C03585=1025.181,-73.447,-90.528,166.772,46.649,158.523
C03586=1025.175,-73.697,-90.517,166.769,46.652,158.524
C03587=1025.169,-73.946,-90.506,166.767,46.655,158.524
C03588=1025.164,-74.196,-90.495,166.763,46.657,158.524
C03589=1025.158,-74.446,-90.485,166.761,46.660,158.524
C03590=1025.152,-74.695,-90.475,166.758,46.663,158.524
C03591=1025.146,-74.945,-90.463,166.755,46.666,158.524
C03592=1025.140,-75.195,-90.452,166.752,46.669,158.525
C03593=1025.135,-75.445,-90.442,166.749,46.672,158.525
C03594=1025.129,-75.694,-90.431,166.746,46.675,158.525
C03595=1025.123,-75.944,-90.421,166.743,46.677,158.525
C03596=1025.117,-76.194,-90.411,166.740,46.680,158.525
C03597=1025.111,-76.443,-90.400,166.737,46.684,158.525
C03598=1025.105,-76.693,-90.389,166.734,46.686,158.525
C03599=1025.099,-76.943,-90.378,166.731,46.689,158.526
C03600=1025.093,-77.193,-90.368,166.728,46.692,158.526
C03601=1025.087,-77.442,-90.358,166.725,46.695,158.526
C03602=1025.082,-77.692,-90.347,166.722,46.698,158.526
C03603=1025.076,-77.942,-90.336,166.719,46.701,158.526
C03604=1025.070,-78.191,-90.326,166.717,46.703,158.526
C03605=1025.064,-78.441,-90.316,166.713,46.707,158.526
C03606=1025.059,-78.690,-90.305,166.710,46.709,158.526
C03607=1025.053,-78.940,-90.294,166.708,46.712,158.527
C03608=1025.047,-79.190,-90.284,166.704,46.715,158.527
C03609=1025.042,-79.440,-90.273,166.701,46.718,158.527
C03610=1025.035,-79.689,-90.263,166.699,46.721,158.527
C03611=1025.029,-79.940,-90.252,166.695,46.724,158.527
C03612=1025.023,-80.189,-90.242,166.692,46.726,158.527
C03613=1025.018,-80.439,-90.231,166.690,46.729,158.527
C03614=1025.011,-80.688,-90.221,166.686,46.732,158.528
C03615=1025.006,-80.938,-90.211,166.683,46.735,158.528
C03616=1025.000,-81.188,-90.201,166.680,46.738,158.528
C03617=1024.994,-81.438,-90.191,166.678,46.741,158.528
C03618=1024.988,-81.688,-90.181,166.674,46.744,158.528
C03619=1024.982,-81.937,-90.170,166.671,46.747,158.528
C03620=1024.976,-82.187,-90.160,166.668,46.750,158.528
C03621=1024.970,-82.436,-90.150,166.666,46.753,158.529
C03622=1024.964,-82.686,-90.140,166.662,46.756,158.529
C03623=1024.959,-82.936,-90.130,166.659,46.759,158.529
C03624=1024.952,-83.185,-90.120,166.657,46.762,158.529
C03625=1024.947,-83.436,-90.109,166.653,46.765,158.529
C03626=1024.941,-83.685,-90.099,166.650,46.768,158.529
C03627=1024.935,-83.935,-90.089,166.647,46.771,158.530
C03628=1024.929,-84.185,-90.079,166.645,46.774,158.530
C03629=1024.923,-84.434,-90.069,166.641,46.777,158.530
C03630=1024.915,-84.787,-90.055,166.637,46.781,158.530
C03631=1024.906,-85.139,-90.040,166.632,46.785,158.530
C03632=1024.899,-85.491,-90.026,166.629,46.790,158.531
C03633=1024.890,-85.842,-90.012,166.625,46.794,158.531
C03634=1024.884,-86.093,-90.002,166.621,46.797,158.531
C03635=1024.878,-86.342,-89.992,166.618,46.800,158.531
C03636=1024.873,-86.592,-89.981,166.616,46.803,158.531
C03637=1024.866,-86.842,-89.972,166.612,46.806,158.532
C03638=1024.861,-87.092,-89.962,166.609,46.809,158.532
C03639=1024.855,-87.342,-89.952,166.606,46.812,158.532
C03640=1024.849,-87.591,-89.941,166.603,46.814,158.532
C03641=1024.843,-87.840,-89.932,166.600,46.817,158.532
C03642=1024.838,-88.090,-89.922,166.597,46.820,158.532
C03643=1024.832,-88.340,-89.912,166.595,46.823,158.532
C03644=1024.826,-88.590,-89.902,166.591,46.826,158.532
C03645=1024.820,-88.839,-89.892,166.588,46.829,158.533
C03646=1024.815,-89.089,-89.882,166.585,46.833,158.533
C03647=1024.808,-89.339,-89.872,166.583,46.835,158.533
C03648=1024.804,-89.589,-89.862,166.579,46.838,158.533
C03649=1024.797,-89.838,-89.853,166.576,46.842,158.533
C03650=1024.792,-90.088,-89.842,166.574,46.844,158.533
C03651=1024.785,-90.338,-89.832,166.571,46.847,158.534
C03652=1024.780,-90.588,-89.822,166.567,46.850,158.534
C03653=1024.774,-90.838,-89.812,166.564,46.853,158.534
C03654=1024.769,-91.087,-89.803,166.561,46.856,158.534
C03655=1024.763,-91.337,-89.793,166.558,46.859,158.534
C03656=1024.757,-91.587,-89.783,166.555,46.862,158.534
C03657=1024.751,-91.837,-89.773,166.552,46.865,158.534
C03658=1024.747,-92.052,-89.764,166.549,46.868,158.534
C03659=1024.741,-92.268,-89.756,166.547,46.870,158.535
C03660=1024.737,-92.483,-89.747,166.545,46.873,158.535
C03661=1024.731,-92.699,-89.739,166.542,46.875,158.535
C03662=1024.727,-92.914,-89.731,166.539,46.878,158.535
C03663=1024.722,-93.129,-89.722,166.536,46.880,158.535
C03664=1024.717,-93.345,-89.714,166.534,46.883,158.535
C03665=1024.712,-93.560,-89.705,166.532,46.885,158.535
C03666=1024.706,-93.810,-89.696,166.528,46.888,158.535
C03667=1024.701,-94.060,-89.686,166.525,46.891,158.536
C03668=1024.695,-94.309,-89.676,166.523,46.894,158.536
C03669=1024.690,-94.559,-89.666,166.520,46.897,158.536
C03670=1024.683,-94.809,-89.656,166.516,46.900,158.536
C03671=1024.677,-95.059,-89.646,166.514,46.902,158.536
C03672=1024.673,-95.309,-89.637,166.510,46.905,158.536
C03673=1024.666,-95.558,-89.628,166.507,46.909,158.536
C03674=1024.661,-95.808,-89.618,166.504,46.912,158.536
C03675=1024.655,-96.058,-89.608,166.502,46.914,158.537
C03676=1024.650,-96.308,-89.598,166.498,46.918,158.537
C03677=1024.644,-96.557,-89.589,166.495,46.921,158.537
C03678=1024.639,-96.807,-89.579,166.493,46.923,158.537
C03679=1024.633,-97.057,-89.569,166.489,46.926,158.537
C03680=1024.627,-97.307,-89.559,166.486,46.929,158.537
C03681=1024.622,-97.556,-89.550,166.483,46.932,158.537
C03682=1024.616,-97.806,-89.540,166.481,46.935,158.538
C03683=1024.610,-98.056,-89.530,166.477,46.938,158.538
C03684=1024.605,-98.306,-89.522,166.474,46.941,158.538
C03685=1024.599,-98.555,-89.512,166.471,46.944,158.538
C03686=1024.593,-98.805,-89.503,166.469,46.947,158.538
C03687=1024.587,-99.054,-89.493,166.465,46.950,158.538
C03688=1024.582,-99.304,-89.483,166.462,46.953,158.538
C03689=1024.576,-99.555,-89.474,166.459,46.956,158.539
C03690=1024.570,-99.804,-89.465,166.455,46.959,158.539
C03691=1024.564,-100.054,-89.456,166.453,46.963,158.539
C03692=1024.558,-100.303,-89.446,166.450,46.966,158.539
C03693=1024.553,-100.553,-89.438,166.447,46.969,158.539
C03694=1024.546,-100.838,-89.426,166.444,46.972,158.539
C03695=1024.539,-101.125,-89.415,166.440,46.976,158.540
C03696=1024.533,-101.411,-89.405,166.436,46.979,158.540
C03697=1024.526,-101.696,-89.394,166.433,46.983,158.540
C03698=1024.521,-101.947,-89.385,166.430,46.986,158.540
C03699=1024.516,-102.196,-89.376,166.427,46.989,158.540
C03700=1024.509,-102.445,-89.366,166.425,46.992,158.541
C03701=1024.504,-102.695,-89.358,166.421,46.995,158.541
C03702=1024.498,-102.945,-89.348,166.418,46.998,158.541
C03703=1024.492,-103.194,-89.339,166.415,47.001,158.541
C03704=1024.487,-103.445,-89.329,166.412,47.004,158.541
C03705=1024.482,-103.694,-89.320,166.409,47.007,158.541
C03706=1024.476,-103.944,-89.311,166.406,47.010,158.541
C03707=1024.470,-104.194,-89.302,166.403,47.014,158.541
C03708=1024.464,-104.443,-89.293,166.400,47.017,158.542
C03709=1024.458,-104.694,-89.284,166.397,47.019,158.542
C03710=1024.453,-104.943,-89.275,166.394,47.023,158.542
C03711=1024.447,-105.193,-89.265,166.391,47.026,158.542
C03712=1024.442,-105.443,-89.256,166.388,47.029,158.542
C03713=1024.436,-105.693,-89.247,166.384,47.032,158.542
C03714=1024.430,-105.942,-89.238,166.382,47.035,158.543
C03715=1024.425,-106.193,-89.229,166.379,47.038,158.543
C03716=1024.419,-106.442,-89.220,166.375,47.041,158.543
C03717=1024.413,-106.692,-89.211,166.372,47.044,158.543
C03718=1024.408,-106.941,-89.202,166.370,47.047,158.543
C03719=1024.402,-107.191,-89.193,166.367,47.050,158.543
C03720=1024.396,-107.441,-89.184,166.363,47.053,158.543
C03721=1024.392,-107.691,-89.175,166.360,47.056,158.543
C03722=1024.385,-107.940,-89.166,166.357,47.059,158.544
C03723=1024.379,-108.190,-89.157,166.355,47.062,158.544
C03724=1024.374,-108.440,-89.148,166.352,47.066,158.544
C03725=1024.368,-108.689,-89.139,166.348,47.069,158.544
C03726=1024.362,-108.940,-89.130,166.345,47.072,158.544
C03727=1024.357,-109.189,-89.121,166.342,47.075,158.544
C03728=1024.351,-109.439,-89.112,166.339,47.078,158.545
C03729=1024.345,-109.689,-89.104,166.336,47.081,158.545
C03730=1024.340,-109.938,-89.095,166.333,47.084,158.545
C03731=1024.334,-110.189,-89.086,166.330,47.087,158.545
C03732=1024.329,-110.438,-89.077,166.327,47.091,158.545
C03733=1024.323,-110.688,-89.068,166.324,47.094,158.545
C03734=1024.317,-110.938,-89.059,166.321,47.097,158.546
C03735=1024.312,-111.187,-89.051,166.318,47.100,158.546
C03736=1024.306,-111.437,-89.041,166.315,47.103,158.546
C03737=1024.301,-111.687,-89.033,166.312,47.106,158.546
C03738=1024.295,-111.937,-89.024,166.308,47.110,158.546
C03739=1024.289,-112.187,-89.015,166.306,47.112,158.546
C03740=1024.283,-112.436,-89.007,166.303,47.116,158.546
C03741=1024.278,-112.686,-88.998,166.300,47.119,158.547
C03742=1024.272,-112.936,-88.989,166.297,47.122,158.547
C03743=1024.267,-113.186,-88.981,166.293,47.126,158.547
C03744=1024.261,-113.435,-88.972,166.291,47.128,158.547
C03745=1024.255,-113.685,-88.963,166.288,47.132,158.547
C03746=1024.250,-113.935,-88.954,166.285,47.135,158.547
C03747=1024.245,-114.185,-88.946,166.281,47.138,158.548
C03748=1024.239,-114.435,-88.937,166.278,47.141,158.548
C03749=1024.233,-114.684,-88.928,166.276,47.144,158.548
C03750=1024.228,-114.934,-88.919,166.273,47.147,158.548
C03751=1024.222,-115.184,-88.911,166.270,47.151,158.548
C03752=1024.216,-115.434,-88.903,166.266,47.154,158.548
C03753=1024.211,-115.683,-88.894,166.263,47.157,158.548
C03754=1024.205,-115.934,-88.885,166.260,47.160,158.549
C03755=1024.200,-116.184,-88.877,166.258,47.163,158.549
C03756=1024.194,-116.433,-88.869,166.254,47.166,158.549
C03757=1024.189,-116.683,-88.860,166.251,47.170,158.549
C03758=1024.182,-116.968,-88.850,166.248,47.173,158.549
C03759=1024.176,-117.253,-88.840,166.244,47.177,158.549
C03760=1024.169,-117.539,-88.830,166.241,47.180,158.550
C03761=1024.163,-117.825,-88.820,166.237,47.184,158.550
C03762=1024.157,-118.074,-88.812,166.235,47.187,158.550
C03763=1024.151,-118.324,-88.804,166.231,47.190,158.550
C03764=1024.146,-118.573,-88.796,166.228,47.193,158.550
C03765=1024.141,-118.823,-88.787,166.225,47.197,158.550
C03766=1024.135,-119.074,-88.778,166.222,47.200,158.551
C03767=1024.129,-119.323,-88.770,166.220,47.203,158.551
C03768=1024.124,-119.573,-88.762,166.216,47.206,158.551
C03769=1024.118,-119.822,-88.753,166.213,47.209,158.551
C03770=1024.113,-120.072,-88.745,166.210,47.213,158.551
C03771=1024.106,-120.322,-88.737,166.207,47.216,158.551
C03772=1024.102,-120.573,-88.729,166.204,47.219,158.552
C03773=1024.096,-120.822,-88.720,166.201,47.222,158.552
C03774=1024.091,-121.072,-88.712,166.198,47.225,158.552
C03775=1024.085,-121.321,-88.704,166.195,47.228,158.552
C03776=1024.080,-121.571,-88.696,166.192,47.232,158.552
C03777=1024.074,-121.822,-88.687,166.189,47.235,158.552
C03778=1024.068,-122.071,-88.679,166.185,47.239,158.552
C03779=1024.063,-122.321,-88.670,166.183,47.241,158.553
C03780=1024.057,-122.570,-88.662,166.180,47.245,158.553
///RCONF 1,0,0,0,0,0,0,0,0,0,0,0,0,0,0,0,0,0,0,0,0,0,0,0
C03781=1024.052,-122.820,-88.655,166.177,47.248,158.553
C03782=1024.046,-123.070,-88.646,166.174,47.252,158.553
C03783=1024.041,-123.320,-88.638,166.170,47.255,158.553
C03784=1024.035,-123.569,-88.630,166.167,47.258,158.553
C03785=1024.029,-123.820,-88.621,166.165,47.261,158.554
C03786=1024.024,-124.069,-88.612,166.162,47.264,158.554
C03787=1024.019,-124.320,-88.605,166.159,47.268,158.554
C03788=1024.013,-124.569,-88.597,166.155,47.271,158.554
C03789=1024.008,-124.819,-88.588,166.152,47.274,158.554
C03790=1024.002,-125.068,-88.580,166.149,47.277,158.554
C03791=1023.997,-125.319,-88.573,166.147,47.281,158.555
C03792=1023.991,-125.568,-88.565,166.144,47.284,158.555
C03793=1023.985,-125.818,-88.556,166.140,47.287,158.555
C03794=1023.981,-126.068,-88.549,166.137,47.290,158.555
C03795=1023.975,-126.317,-88.541,166.134,47.294,158.555
C03796=1023.969,-126.567,-88.532,166.131,47.297,158.555
C03797=1023.963,-126.818,-88.525,166.128,47.300,158.555
C03798=1023.958,-127.068,-88.516,166.125,47.303,158.556
C03799=1023.952,-127.317,-88.508,166.123,47.307,158.556
C03800=1023.947,-127.567,-88.500,166.119,47.310,158.556
C03801=1023.941,-127.817,-88.493,166.116,47.313,158.556
C03802=1023.936,-128.066,-88.484,166.113,47.316,158.556
C03803=1023.931,-128.315,-88.476,166.111,47.319,158.556
C03804=1023.926,-128.566,-88.467,166.108,47.320,158.556
C03805=1023.923,-128.815,-88.457,166.104,47.323,158.556
C03806=1023.919,-129.065,-88.446,166.102,47.323,158.556
C03807=1023.917,-129.314,-88.435,166.099,47.325,158.556
C03808=1023.914,-129.564,-88.424,166.097,47.325,158.556
C03809=1023.912,-129.814,-88.411,166.095,47.324,158.555
C03810=1023.912,-130.064,-88.399,166.092,47.323,158.555
C03811=1023.911,-130.313,-88.386,166.090,47.322,158.554
C03812=1023.911,-130.563,-88.371,166.087,47.321,158.554
C03813=1023.911,-130.813,-88.357,166.085,47.318,158.553
C03814=1023.912,-131.063,-88.342,166.084,47.315,158.552
C03815=1023.913,-131.313,-88.326,166.082,47.312,158.552
C03816=1023.915,-131.562,-88.310,166.080,47.308,158.551
C03817=1023.918,-131.811,-88.293,166.078,47.304,158.550
C03818=1023.920,-132.062,-88.276,166.076,47.299,158.549
C03819=1023.925,-132.312,-88.258,166.075,47.294,158.548
C03820=1023.927,-132.562,-88.239,166.073,47.288,158.546
C03821=1023.933,-132.810,-88.220,166.072,47.282,158.545
C03822=1023.637,-132.837,-88.558,166.025,47.565,158.587
C03823=1023.633,-132.587,-88.577,166.026,47.571,158.588
C03824=1023.629,-132.338,-88.595,166.027,47.577,158.589
C03825=1023.625,-132.088,-88.613,166.028,47.582,158.590
C03826=1023.622,-131.838,-88.631,166.030,47.587,158.591
C03827=1023.620,-131.589,-88.648,166.032,47.591,158.592
C03828=1023.618,-131.339,-88.664,166.034,47.595,158.593
C03829=1023.617,-131.088,-88.680,166.036,47.598,158.594
C03830=1023.616,-130.839,-88.695,166.037,47.601,158.594
C03831=1023.615,-130.589,-88.709,166.039,47.603,158.595
C03832=1023.616,-130.340,-88.723,166.042,47.605,158.596
C03833=1023.617,-130.089,-88.737,166.044,47.606,158.596
C03834=1023.618,-129.839,-88.749,166.047,47.607,158.597
C03835=1023.619,-129.590,-88.762,166.049,47.608,158.597
C03836=1023.621,-129.340,-88.773,166.051,47.607,158.597
C03837=1023.624,-129.090,-88.784,166.054,47.606,158.598
C03838=1023.627,-128.841,-88.794,166.057,47.605,158.598
C03839=1023.631,-128.591,-88.805,166.060,47.603,158.598
C03840=1023.635,-128.342,-88.814,166.062,47.601,158.598
C03841=1023.641,-128.092,-88.822,166.065,47.599,158.598
C03842=1023.646,-127.842,-88.831,166.068,47.596,158.598
C03843=1023.651,-127.593,-88.839,166.071,47.592,158.597
C03844=1023.657,-127.343,-88.846,166.074,47.589,158.597
C03845=1023.662,-127.093,-88.855,166.078,47.586,158.597
C03846=1023.668,-126.843,-88.862,166.081,47.582,158.597
C03847=1023.673,-126.593,-88.870,166.084,47.579,158.597
C03848=1023.679,-126.344,-88.878,166.086,47.576,158.597
C03849=1023.684,-126.093,-88.886,166.089,47.572,158.596
C03850=1023.690,-125.844,-88.894,166.092,47.569,158.596
C03851=1023.695,-125.594,-88.902,166.095,47.566,158.596
C03852=1023.700,-125.344,-88.910,166.098,47.562,158.596
C03853=1023.706,-125.095,-88.918,166.102,47.559,158.596
C03854=1023.711,-124.845,-88.926,166.105,47.555,158.596
C03855=1023.717,-124.595,-88.934,166.108,47.552,158.596
C03856=1023.722,-124.345,-88.942,166.111,47.548,158.595
C03857=1023.728,-124.096,-88.950,166.113,47.545,158.595
C03858=1023.734,-123.846,-88.959,166.117,47.542,158.595
C03859=1023.740,-123.596,-88.967,166.120,47.539,158.595
C03860=1023.744,-123.345,-88.975,166.123,47.535,158.595
C03861=1023.750,-123.096,-88.983,166.126,47.532,158.595
C03862=1023.756,-122.846,-88.992,166.129,47.529,158.594
C03863=1023.761,-122.596,-89.000,166.132,47.526,158.594
C03864=1023.767,-122.347,-89.008,166.135,47.522,158.594
C03865=1023.772,-122.097,-89.016,166.138,47.519,158.594
C03866=1023.777,-121.847,-89.024,166.141,47.516,158.594
C03867=1023.783,-121.598,-89.032,166.144,47.513,158.594
C03868=1023.789,-121.347,-89.041,166.147,47.509,158.593
C03869=1023.794,-121.097,-89.049,166.150,47.506,158.593
C03870=1023.800,-120.848,-89.057,166.154,47.503,158.593
C03871=1023.806,-120.598,-89.066,166.157,47.500,158.593
C03872=1023.811,-120.349,-89.074,166.159,47.496,158.593
C03873=1023.816,-120.099,-89.083,166.162,47.493,158.593
C03874=1023.823,-119.849,-89.091,166.165,47.490,158.592
C03875=1023.828,-119.599,-89.099,166.168,47.487,158.592
C03876=1023.833,-119.349,-89.107,166.172,47.483,158.592
C03877=1023.838,-119.099,-89.116,166.175,47.480,158.592
C03878=1023.844,-118.850,-89.124,166.178,47.476,158.592
C03879=1023.850,-118.600,-89.132,166.181,47.473,158.592
C03880=1023.855,-118.349,-89.141,166.183,47.470,158.592
C03881=1023.861,-118.100,-89.149,166.186,47.467,158.591
C03882=1023.867,-117.850,-89.157,166.190,47.463,158.591
C03883=1023.873,-117.565,-89.167,166.194,47.459,158.591
C03884=1023.879,-117.280,-89.177,166.197,47.456,158.591
C03885=1023.885,-116.995,-89.187,166.200,47.452,158.591
C03886=1023.892,-116.709,-89.197,166.204,47.448,158.590
C03887=1023.897,-116.459,-89.205,166.207,47.445,158.590
C03888=1023.903,-116.210,-89.214,166.210,47.442,158.590
C03889=1023.909,-115.960,-89.222,166.212,47.439,158.590
C03890=1023.915,-115.710,-89.231,166.216,47.436,158.590
C03891=1023.920,-115.460,-89.239,166.219,47.432,158.590
C03892=1023.925,-115.210,-89.247,166.222,47.429,158.589
C03893=1023.931,-114.960,-89.256,166.225,47.426,158.589
C03894=1023.937,-114.711,-89.264,166.228,47.423,158.589
C03895=1023.942,-114.461,-89.273,166.231,47.419,158.589
C03896=1023.948,-114.211,-89.282,166.233,47.416,158.589
C03897=1023.954,-113.961,-89.291,166.237,47.413,158.589
C03898=1023.959,-113.712,-89.299,166.240,47.410,158.589
C03899=1023.965,-113.461,-89.308,166.243,47.406,158.588
C03900=1023.970,-113.211,-89.317,166.246,47.403,158.588
C03901=1023.975,-112.962,-89.325,166.249,47.400,158.588
C03902=1023.981,-112.712,-89.335,166.252,47.397,158.588
C03903=1023.987,-112.462,-89.343,166.255,47.393,158.588
C03904=1023.992,-112.213,-89.352,166.258,47.390,158.588
C03905=1023.999,-111.962,-89.360,166.261,47.387,158.587
C03906=1024.004,-111.713,-89.369,166.265,47.384,158.587
C03907=1024.009,-111.464,-89.378,166.268,47.381,158.587
C03908=1024.015,-111.213,-89.386,166.271,47.377,158.587
C03909=1024.021,-110.964,-89.396,166.273,47.374,158.587
C03910=1024.026,-110.714,-89.404,166.276,47.371,158.587
C03911=1024.032,-110.464,-89.413,166.280,47.368,158.587
C03912=1024.037,-110.214,-89.421,166.283,47.365,158.586
C03913=1024.043,-109.965,-89.431,166.286,47.361,158.586
C03914=1024.049,-109.715,-89.439,166.289,47.358,158.586
C03915=1024.054,-109.465,-89.448,166.291,47.355,158.586
C03916=1024.060,-109.215,-89.458,166.294,47.352,158.586
C03917=1024.065,-108.966,-89.466,166.298,47.349,158.586
C03918=1024.071,-108.716,-89.475,166.301,47.346,158.585
C03919=1024.077,-108.466,-89.484,166.304,47.342,158.585
C03920=1024.082,-108.216,-89.493,166.307,47.339,158.585
C03921=1024.088,-107.966,-89.502,166.310,47.336,158.585
C03922=1024.094,-107.717,-89.511,166.313,47.333,158.585
C03923=1024.099,-107.466,-89.519,166.316,47.330,158.585
C03924=1024.105,-107.217,-89.529,166.319,47.326,158.585
C03925=1024.111,-106.967,-89.538,166.322,47.323,158.584
C03926=1024.116,-106.718,-89.547,166.325,47.319,158.584
C03927=1024.122,-106.468,-89.555,166.329,47.316,158.584
C03928=1024.128,-106.218,-89.565,166.331,47.313,158.584
C03929=1024.133,-105.969,-89.573,166.334,47.310,158.584
C03930=1024.139,-105.719,-89.583,166.337,47.307,158.584
C03931=1024.145,-105.469,-89.591,166.341,47.304,158.583
C03932=1024.151,-105.219,-89.601,166.344,47.301,158.583
C03933=1024.155,-104.969,-89.610,166.347,47.298,158.583
C03934=1024.161,-104.719,-89.620,166.349,47.295,158.583
C03935=1024.167,-104.470,-89.628,166.352,47.291,158.583
C03936=1024.173,-104.220,-89.638,166.355,47.288,158.583
C03937=1024.178,-103.970,-89.646,166.359,47.285,158.582
C03938=1024.184,-103.720,-89.656,166.362,47.282,158.582
C03939=1024.190,-103.471,-89.665,166.364,47.279,158.582
C03940=1024.195,-103.221,-89.674,166.367,47.276,158.582
C03941=1024.201,-102.971,-89.683,166.371,47.273,158.582
C03942=1024.206,-102.721,-89.692,166.374,47.270,158.582
C03943=1024.213,-102.471,-89.702,166.377,47.266,158.582
C03944=1024.218,-102.222,-89.711,166.380,47.263,158.582
C03945=1024.224,-101.972,-89.720,166.383,47.260,158.581
C03946=1024.229,-101.722,-89.730,166.386,47.257,158.581
C03947=1024.236,-101.437,-89.740,166.390,47.253,158.581
C03948=1024.242,-101.151,-89.751,166.393,47.249,158.581
C03949=1024.249,-100.865,-89.762,166.396,47.246,158.581
C03950=1024.256,-100.579,-89.772,166.400,47.242,158.580
C03951=1024.260,-100.330,-89.781,166.402,47.239,158.580
C03952=1024.267,-100.080,-89.791,166.406,47.236,158.580
C03953=1024.273,-99.830,-89.800,166.409,47.233,158.580
C03954=1024.278,-99.581,-89.809,166.412,47.230,158.580
C03955=1024.284,-99.331,-89.819,166.415,47.227,158.580
C03956=1024.290,-99.082,-89.828,166.419,47.224,158.580
C03957=1024.295,-98.831,-89.837,166.421,47.220,158.579
C03958=1024.301,-98.581,-89.847,166.424,47.217,158.579
C03959=1024.307,-98.332,-89.856,166.427,47.214,158.579
C03960=1024.313,-98.082,-89.866,166.430,47.211,158.579
C03961=1024.319,-97.832,-89.874,166.434,47.208,158.579
C03962=1024.324,-97.582,-89.884,166.436,47.205,158.579
C03963=1024.330,-97.333,-89.894,166.439,47.202,158.578
C03964=1024.335,-97.082,-89.904,166.442,47.199,158.578
C03965=1024.341,-96.833,-89.913,166.446,47.196,158.578
C03966=1024.346,-96.583,-89.923,166.448,47.193,158.578
C03967=1024.352,-96.333,-89.933,166.451,47.190,158.578
C03968=1024.358,-96.084,-89.942,166.454,47.187,158.578
C03969=1024.363,-95.834,-89.952,166.457,47.183,158.578
C03970=1024.370,-95.584,-89.962,166.460,47.181,158.577
C03971=1024.374,-95.335,-89.972,166.463,47.177,158.577
C03972=1024.381,-95.085,-89.981,166.466,47.174,158.577
C03973=1024.386,-94.835,-89.991,166.470,47.172,158.577
C03974=1024.391,-94.585,-90.000,166.472,47.169,158.577
C03975=1024.397,-94.335,-90.010,166.475,47.166,158.577
C03976=1024.403,-94.086,-90.020,166.478,47.163,158.577
C03977=1024.408,-93.836,-90.029,166.482,47.160,158.577
C03978=1024.414,-93.587,-90.040,166.485,47.157,158.576
C03979=1024.420,-93.337,-90.050,166.487,47.154,158.576
C03980=1024.426,-93.087,-90.059,166.490,47.151,158.576
C03981=1024.431,-92.838,-90.069,166.494,47.148,158.576
C03982=1024.437,-92.588,-90.079,166.497,47.144,158.576
C03983=1024.443,-92.338,-90.088,166.499,47.142,158.576
C03984=1024.448,-92.088,-90.098,166.502,47.138,158.576
C03985=1024.454,-91.839,-90.108,166.506,47.135,158.575
C03986=1024.459,-91.589,-90.118,166.509,47.132,158.575
C03987=1024.466,-91.339,-90.127,166.511,47.129,158.575
C03988=1024.471,-91.089,-90.138,166.514,47.126,158.575
C03989=1024.477,-90.839,-90.147,166.518,47.123,158.575
C03990=1024.482,-90.590,-90.157,166.521,47.120,158.575
C03991=1024.488,-90.340,-90.166,166.523,47.117,158.574
C03992=1024.494,-90.090,-90.177,166.526,47.114,158.574
C03993=1024.500,-89.841,-90.187,166.530,47.111,158.574
C03994=1024.505,-89.590,-90.197,166.533,47.108,158.574
C03995=1024.511,-89.341,-90.206,166.535,47.105,158.574
C03996=1024.516,-89.091,-90.216,166.538,47.102,158.574
C03997=1024.523,-88.841,-90.226,166.542,47.099,158.574
C03998=1024.528,-88.592,-90.237,166.545,47.096,158.573
C03999=1024.535,-88.342,-90.246,166.548,47.093,158.573
C04000=1024.540,-88.092,-90.257,166.550,47.090,158.573
C04001=1024.546,-87.843,-90.266,166.554,47.087,158.573
C04002=1024.551,-87.593,-90.276,166.557,47.084,158.573
C04003=1024.557,-87.344,-90.286,166.560,47.081,158.573
C04004=1024.563,-87.094,-90.296,166.562,47.078,158.572
C04005=1024.569,-86.844,-90.306,166.566,47.075,158.572
C04006=1024.575,-86.594,-90.316,166.569,47.072,158.572
C04007=1024.581,-86.344,-90.326,166.572,47.068,158.572
C04008=1024.586,-86.094,-90.337,166.574,47.066,158.572
C04009=1024.593,-85.845,-90.346,166.578,47.062,158.572
C04010=1024.597,-85.595,-90.356,166.581,47.059,158.572
C04011=1024.605,-85.312,-90.368,166.584,47.056,158.571
C04012=1024.611,-85.028,-90.379,166.588,47.052,158.571
C04013=1024.618,-84.744,-90.391,166.591,47.048,158.571
C04014=1024.625,-84.460,-90.402,166.594,47.045,158.571
C04015=1024.630,-84.212,-90.412,166.598,47.042,158.571
C04016=1024.636,-83.962,-90.422,166.601,47.039,158.571
C04017=1024.642,-83.712,-90.432,166.603,47.036,158.570
C04018=1024.648,-83.462,-90.443,166.606,47.033,158.570
C04019=1024.654,-83.212,-90.452,166.610,47.030,158.570
C04020=1024.659,-82.963,-90.463,166.613,47.027,158.570
C04021=1024.666,-82.713,-90.473,166.616,47.024,158.570
C04022=1024.671,-82.463,-90.483,166.618,47.021,158.570
C04023=1024.678,-82.214,-90.493,166.621,47.017,158.569
C04024=1024.683,-81.964,-90.503,166.625,47.014,158.569
C04025=1024.689,-81.714,-90.514,166.628,47.011,158.569
C04026=1024.695,-81.464,-90.524,166.630,47.008,158.569
C04027=1024.701,-81.215,-90.533,166.633,47.005,158.569
C04028=1024.707,-80.965,-90.544,166.637,47.002,158.569
C04029=1024.713,-80.715,-90.554,166.640,46.999,158.568
C04030=1024.719,-80.466,-90.565,166.643,46.996,158.568
C04031=1024.725,-80.216,-90.574,166.645,46.993,158.568
C04032=1024.731,-79.966,-90.585,166.649,46.990,158.568
C04033=1024.737,-79.716,-90.596,166.652,46.987,158.568
C04034=1024.742,-79.466,-90.606,166.655,46.984,158.568
C04035=1024.748,-79.216,-90.617,166.657,46.981,158.567
C04036=1024.754,-78.967,-90.627,166.661,46.978,158.567
C04037=1024.760,-78.717,-90.637,166.664,46.975,158.567
C04038=1024.765,-78.467,-90.648,166.666,46.972,158.567
C04039=1024.773,-78.159,-90.661,166.670,46.969,158.567
C04040=1024.779,-77.850,-90.674,166.673,46.965,158.567
C04041=1024.786,-77.541,-90.687,166.678,46.962,158.567
C04042=1024.794,-77.232,-90.700,166.682,46.957,158.566
C04043=1024.800,-76.983,-90.710,166.684,46.955,158.566
C04044=1024.806,-76.734,-90.721,166.687,46.952,158.566
C04045=1024.811,-76.484,-90.731,166.690,46.948,158.566
C04046=1024.817,-76.234,-90.742,166.693,46.946,158.566
C04047=1024.823,-75.984,-90.753,166.696,46.943,158.566
C04048=1024.830,-75.734,-90.763,166.700,46.940,158.566
C04049=1024.835,-75.485,-90.774,166.703,46.937,158.565
C04050=1024.841,-75.235,-90.785,166.705,46.934,158.565
C04051=1024.847,-74.985,-90.795,166.708,46.931,158.565
C04052=1024.852,-74.735,-90.806,166.712,46.928,158.565
C04053=1024.858,-74.486,-90.817,166.714,46.925,158.565
C04054=1024.865,-74.236,-90.827,166.717,46.922,158.565
C04055=1024.871,-73.987,-90.838,166.720,46.919,158.564
C04056=1024.876,-73.736,-90.849,166.723,46.916,158.564
C04057=1024.881,-73.487,-90.860,166.726,46.914,158.564
C04058=1024.887,-73.237,-90.871,166.729,46.911,158.564
C04059=1024.893,-72.988,-90.882,166.732,46.908,158.564
C04060=1024.899,-72.738,-90.892,166.735,46.906,158.564
C04061=1024.904,-72.489,-90.903,166.737,46.903,158.564
C04062=1024.911,-72.239,-90.915,166.741,46.900,158.564
C04063=1024.916,-71.989,-90.925,166.744,46.897,158.563
C04064=1024.922,-71.740,-90.936,166.746,46.894,158.563
C04065=1024.928,-71.490,-90.947,166.750,46.891,158.563
C04066=1024.932,-71.240,-90.958,166.753,46.888,158.563
C04067=1024.939,-70.989,-90.969,166.755,46.886,158.563
C04068=1024.945,-70.740,-90.980,166.758,46.882,158.563
C04069=1024.950,-70.490,-90.991,166.761,46.880,158.563
C04070=1024.956,-70.241,-91.002,166.764,46.877,158.562
C04071=1024.961,-70.005,-91.012,166.767,46.874,158.562
C04072=1024.967,-69.769,-91.022,166.770,46.872,158.562
C04073=1024.972,-69.533,-91.033,166.772,46.869,158.562
C04074=1024.978,-69.296,-91.044,166.775,46.866,158.562
C04075=1024.983,-69.060,-91.054,166.778,46.864,158.562
C04076=1024.989,-68.824,-91.064,166.781,46.861,158.562
C04077=1024.994,-68.588,-91.075,166.784,46.859,158.562
C04078=1024.999,-68.352,-91.085,166.787,46.856,158.562
C04079=1025.006,-68.103,-91.097,166.789,46.853,158.561
C04080=1025.012,-67.853,-91.108,166.793,46.850,158.561
C04081=1025.018,-67.604,-91.119,166.795,46.847,158.561
C04082=1025.023,-67.354,-91.130,166.798,46.845,158.561
C04083=1025.030,-67.104,-91.141,166.802,46.842,158.561
C04084=1025.035,-66.855,-91.152,166.804,46.839,158.561
C04085=1025.040,-66.605,-91.164,166.807,46.836,158.560
C04086=1025.046,-66.355,-91.175,166.810,46.833,158.560
C04087=1025.052,-66.105,-91.186,166.813,46.830,158.560
C04088=1025.058,-65.856,-91.197,166.816,46.827,158.560
C04089=1025.064,-65.606,-91.208,166.818,46.825,158.560
C04090=1025.071,-65.356,-91.219,166.822,46.821,158.560
///RCONF 1,0,0,1,0,0,0,0,0,0,0,0,0,0,0,0,0,0,0,0,0,0,0,0
C04091=1025.076,-65.107,-91.230,166.825,46.818,158.560
C04092=1025.081,-64.857,-91.242,166.827,46.816,158.560
C04093=1025.088,-64.607,-91.253,166.831,46.813,158.559
C04094=1025.093,-64.358,-91.264,166.834,46.810,158.559
C04095=1025.099,-64.108,-91.275,166.836,46.807,158.559
C04096=1025.106,-63.858,-91.286,166.839,46.804,158.559
C04097=1025.112,-63.609,-91.298,166.843,46.801,158.559
C04098=1025.117,-63.359,-91.309,166.845,46.799,158.559
C04099=1025.123,-63.109,-91.320,166.848,46.796,158.558
C04100=1025.129,-62.859,-91.331,166.851,46.793,158.558
C04101=1025.135,-62.610,-91.343,166.854,46.790,158.558
C04102=1025.141,-62.360,-91.354,166.857,46.787,158.558
C04103=1025.147,-62.111,-91.365,166.859,46.784,158.558
C04104=1025.153,-61.861,-91.376,166.863,46.781,158.558
C04105=1025.158,-61.612,-91.388,166.866,46.779,158.558
C04106=1025.165,-61.361,-91.400,166.869,46.776,158.557
C04107=1025.170,-61.112,-91.411,166.872,46.773,158.557
C04108=1025.176,-60.862,-91.421,166.875,46.770,158.557
C04109=1025.183,-60.613,-91.433,166.877,46.767,158.557
C04110=1025.189,-60.363,-91.444,166.881,46.764,158.557
C04111=1025.194,-60.113,-91.456,166.883,46.761,158.557
C04112=1025.200,-59.864,-91.468,166.886,46.758,158.556
C04113=1025.207,-59.614,-91.479,166.890,46.756,158.556
C04114=1025.212,-59.364,-91.490,166.892,46.753,158.556
C04115=1025.219,-59.115,-91.502,166.895,46.750,158.556
C04116=1025.224,-58.865,-91.513,166.898,46.747,158.556
C04117=1025.230,-58.615,-91.524,166.901,46.744,158.556
C04118=1025.236,-58.366,-91.536,166.904,46.741,158.555
C04119=1025.243,-58.116,-91.547,166.907,46.738,158.555
C04120=1025.248,-57.866,-91.558,166.909,46.735,158.555
C04121=1025.255,-57.617,-91.570,166.913,46.732,158.555
C04122=1025.260,-57.367,-91.582,166.915,46.729,158.555
C04123=1025.266,-57.117,-91.593,166.918,46.727,158.555
C04124=1025.272,-56.868,-91.604,166.922,46.724,158.555
C04125=1025.279,-56.618,-91.616,166.924,46.721,158.554
C04126=1025.285,-56.369,-91.627,166.927,46.718,158.554
C04127=1025.290,-56.118,-91.639,166.930,46.715,158.554
C04128=1025.297,-55.869,-91.651,166.933,46.712,158.554
C04129=1025.303,-55.619,-91.662,166.936,46.709,158.554
C04130=1025.309,-55.370,-91.674,166.939,46.706,158.554
C04131=1025.315,-55.120,-91.685,166.941,46.703,158.553
C04132=1025.320,-54.870,-91.696,166.945,46.700,158.553
C04133=1025.327,-54.621,-91.708,166.947,46.697,158.553
C04134=1025.333,-54.370,-91.719,166.950,46.694,158.553
C04135=1025.339,-54.122,-91.731,166.954,46.691,158.553
C04136=1025.346,-53.871,-91.742,166.956,46.688,158.552
C04137=1025.351,-53.622,-91.754,166.959,46.686,158.552
C04138=1025.357,-53.372,-91.766,166.963,46.683,158.552
C04139=1025.364,-53.092,-91.779,166.966,46.679,158.552
C04140=1025.372,-52.812,-91.792,166.969,46.676,158.552
C04141=1025.378,-52.532,-91.805,166.972,46.673,158.552
C04142=1025.384,-52.252,-91.818,166.975,46.669,158.551
C04143=1025.391,-52.001,-91.830,166.978,46.666,158.551
C04144=1025.397,-51.752,-91.842,166.981,46.663,158.551
C04145=1025.403,-51.503,-91.853,166.984,46.660,158.551
C04146=1025.410,-51.253,-91.864,166.987,46.657,158.551
C04147=1025.416,-51.003,-91.877,166.989,46.655,158.550
C04148=1025.421,-50.753,-91.888,166.993,46.651,158.550
C04149=1025.427,-50.504,-91.900,166.995,46.649,158.550
C04150=1025.434,-50.254,-91.912,166.998,46.646,158.550
C04151=1025.439,-50.004,-91.924,167.001,46.643,158.550
C04152=1025.446,-49.755,-91.936,167.004,46.641,158.550
C04153=1025.452,-49.505,-91.948,167.006,46.638,158.550
C04154=1025.457,-49.256,-91.961,167.010,46.635,158.549
C04155=1025.464,-49.006,-91.972,167.013,46.632,158.549
C04156=1025.469,-48.756,-91.984,167.016,46.630,158.549
C04157=1025.475,-48.507,-91.996,167.019,46.627,158.549
C04158=1025.481,-48.257,-92.008,167.021,46.624,158.549
C04159=1025.486,-48.008,-92.021,167.025,46.622,158.549
C04160=1025.493,-47.758,-92.033,167.027,46.619,158.549
C04161=1025.499,-47.507,-92.044,167.030,46.616,158.548
C04162=1025.505,-47.258,-92.056,167.032,46.613,158.548
C04163=1025.511,-47.009,-92.069,167.036,46.611,158.548
C04164=1025.516,-46.759,-92.081,167.038,46.608,158.548
C04165=1025.523,-46.509,-92.093,167.041,46.605,158.548
C04166=1025.528,-46.260,-92.105,167.044,46.602,158.548
C04167=1025.535,-46.011,-92.117,167.047,46.600,158.548
C04168=1025.541,-45.761,-92.130,167.049,46.597,158.547
C04169=1025.546,-45.511,-92.141,167.053,46.594,158.547
C04170=1025.553,-45.261,-92.153,167.055,46.591,158.547
C04171=1025.559,-45.011,-92.166,167.058,46.588,158.547
C04172=1025.565,-44.762,-92.178,167.061,46.586,158.547
C04173=1025.571,-44.513,-92.190,167.064,46.583,158.547
C04174=1025.576,-44.263,-92.202,167.067,46.580,158.546
C04175=1025.583,-44.013,-92.214,167.070,46.577,158.546
C04176=1025.589,-43.763,-92.227,167.073,46.575,158.546
C04177=1025.594,-43.514,-92.239,167.075,46.572,158.546
C04178=1025.601,-43.265,-92.251,167.079,46.569,158.546
C04179=1025.607,-43.015,-92.264,167.081,46.566,158.546
C04180=1025.613,-42.765,-92.276,167.084,46.563,158.545
C04181=1025.619,-42.515,-92.288,167.087,46.561,158.545
C04182=1025.625,-42.266,-92.300,167.090,46.558,158.545
C04183=1025.631,-42.016,-92.312,167.092,46.555,158.545
C04184=1025.637,-41.767,-92.325,167.095,46.552,158.545
C04185=1025.643,-41.517,-92.337,167.098,46.549,158.545
C04186=1025.650,-41.267,-92.349,167.101,46.547,158.545
C04187=1025.655,-41.018,-92.362,167.103,46.544,158.544
C04188=1025.661,-40.768,-92.374,167.107,46.541,158.544
C04189=1025.668,-40.518,-92.386,167.109,46.538,158.544
C04190=1025.674,-40.269,-92.399,167.112,46.535,158.544
C04191=1025.679,-40.019,-92.411,167.116,46.532,158.544
C04192=1025.686,-39.769,-92.423,167.118,46.530,158.544
C04193=1025.692,-39.519,-92.436,167.121,46.527,158.543
C04194=1025.698,-39.271,-92.448,167.124,46.524,158.543
C04195=1025.704,-39.021,-92.461,167.127,46.521,158.543
C04196=1025.710,-38.771,-92.473,167.129,46.519,158.543
C04197=1025.716,-38.521,-92.486,167.133,46.516,158.543
C04198=1025.722,-38.271,-92.498,167.135,46.513,158.543
C04199=1025.728,-38.022,-92.511,167.137,46.511,158.542
C04200=1025.734,-37.772,-92.524,167.141,46.508,158.542
C04201=1025.739,-37.523,-92.536,167.143,46.506,158.542
C04202=1025.745,-37.273,-92.549,167.146,46.503,158.542
C04203=1025.753,-36.993,-92.563,167.150,46.500,158.542
C04204=1025.759,-36.713,-92.577,167.153,46.496,158.542
C04205=1025.766,-36.433,-92.592,167.155,46.494,158.541
C04206=1025.773,-36.154,-92.606,167.158,46.491,158.541
C04207=1025.779,-35.904,-92.618,167.162,46.488,158.541
C04208=1025.785,-35.654,-92.631,167.164,46.486,158.541
C04209=1025.791,-35.404,-92.644,167.167,46.482,158.541
C04210=1025.798,-35.155,-92.656,167.170,46.480,158.541
C04211=1025.803,-34.906,-92.669,167.173,46.477,158.541
C04212=1025.809,-34.656,-92.681,167.175,46.475,158.540
C04213=1025.815,-34.407,-92.694,167.179,46.472,158.540
C04214=1025.821,-34.157,-92.707,167.181,46.469,158.540
C04215=1025.827,-33.907,-92.719,167.183,46.467,158.540
C04216=1025.833,-33.658,-92.733,167.187,46.464,158.540
C04217=1025.839,-33.408,-92.745,167.189,46.461,158.540
C04218=1025.845,-33.159,-92.758,167.193,46.459,158.539
C04219=1025.851,-32.909,-92.771,167.195,46.456,158.539
C04220=1025.857,-32.659,-92.784,167.198,46.453,158.539
C04221=1025.863,-32.410,-92.797,167.200,46.450,158.539
C04222=1025.869,-32.160,-92.809,167.204,46.448,158.539
C04223=1025.876,-31.911,-92.822,167.206,46.445,158.539
C04224=1025.882,-31.661,-92.835,167.209,46.442,158.538
C04225=1025.888,-31.411,-92.847,167.212,46.439,158.538
C04226=1025.894,-31.162,-92.860,167.214,46.437,158.538
C04227=1025.900,-30.912,-92.873,167.217,46.434,158.538
C04228=1025.906,-30.663,-92.886,167.220,46.431,158.538
C04229=1025.912,-30.413,-92.899,167.223,46.428,158.538
C04230=1025.918,-30.164,-92.912,167.226,46.426,158.538
C04231=1025.924,-29.914,-92.925,167.229,46.423,158.537
C04232=1025.930,-29.665,-92.938,167.231,46.420,158.537
C04233=1025.936,-29.415,-92.950,167.234,46.417,158.537
C04234=1025.943,-29.165,-92.964,167.237,46.414,158.537
C04235=1025.948,-28.916,-92.976,167.240,46.412,158.537
C04236=1025.955,-28.666,-92.990,167.242,46.409,158.536
C04237=1025.961,-28.416,-93.002,167.245,46.406,158.536
C04238=1025.967,-28.166,-93.016,167.248,46.403,158.536
C04239=1025.973,-27.917,-93.028,167.250,46.401,158.536
C04240=1025.980,-27.668,-93.041,167.254,46.398,158.536
C04241=1025.986,-27.418,-93.054,167.256,46.396,158.536
C04242=1025.992,-27.168,-93.067,167.259,46.393,158.535
C04243=1025.998,-26.919,-93.081,167.262,46.390,158.535
C04244=1026.004,-26.669,-93.093,167.264,46.388,158.535
C04245=1026.010,-26.420,-93.106,167.267,46.385,158.535
C04246=1026.016,-26.170,-93.120,167.270,46.383,158.535
C04247=1026.021,-25.920,-93.133,167.273,46.380,158.535
C04248=1026.028,-25.671,-93.146,167.275,46.377,158.534
C04249=1026.034,-25.422,-93.159,167.278,46.375,158.534
C04250=1026.040,-25.172,-93.172,167.281,46.372,158.534
C04251=1026.046,-24.922,-93.186,167.283,46.369,158.534
C04252=1026.052,-24.672,-93.200,167.287,46.367,158.534
C04253=1026.058,-24.423,-93.213,167.289,46.364,158.534
C04254=1026.064,-24.173,-93.225,167.291,46.361,158.533
C04255=1026.070,-23.924,-93.239,167.295,46.359,158.533
C04256=1026.076,-23.674,-93.252,167.297,46.356,158.533
C04257=1026.082,-23.425,-93.266,167.300,46.353,158.533
C04258=1026.088,-23.175,-93.278,167.303,46.351,158.533
C04259=1026.095,-22.925,-93.292,167.305,46.348,158.533
C04260=1026.101,-22.676,-93.305,167.309,46.345,158.533
C04261=1026.106,-22.426,-93.319,167.311,46.343,158.532
C04262=1026.112,-22.176,-93.332,167.313,46.340,158.532
C04263=1026.119,-21.927,-93.345,167.317,46.337,158.532
C04264=1026.125,-21.678,-93.358,167.319,46.335,158.532
C04265=1026.131,-21.428,-93.372,167.322,46.332,158.532
C04266=1026.137,-21.178,-93.386,167.325,46.329,158.532
C04267=1026.144,-20.898,-93.400,167.328,46.326,158.531
C04268=1026.151,-20.617,-93.415,167.331,46.323,158.531
C04269=1026.158,-20.337,-93.430,167.334,46.320,158.531
C04270=1026.165,-20.055,-93.446,167.337,46.317,158.531
C04271=1026.171,-19.806,-93.459,167.340,46.314,158.531
C04272=1026.177,-19.556,-93.472,167.342,46.312,158.530
C04273=1026.182,-19.307,-93.486,167.345,46.310,158.530
C04274=1026.189,-19.057,-93.499,167.348,46.307,158.530
C04275=1026.195,-18.807,-93.513,167.350,46.304,158.530
C04276=1026.202,-18.558,-93.526,167.353,46.301,158.530
C04277=1026.207,-18.309,-93.540,167.356,46.299,158.530
C04278=1026.213,-18.059,-93.553,167.358,46.296,158.529
C04279=1026.220,-17.809,-93.567,167.362,46.293,158.529
C04280=1026.226,-17.560,-93.580,167.364,46.290,158.529
C04281=1026.232,-17.311,-93.594,167.367,46.288,158.529
C04282=1026.238,-17.061,-93.607,167.370,46.285,158.529
C04283=1026.245,-16.811,-93.621,167.372,46.282,158.529
C04284=1026.251,-16.562,-93.634,167.375,46.279,158.528
C04285=1026.256,-16.312,-93.647,167.378,46.277,158.528
C04286=1026.263,-16.062,-93.661,167.380,46.274,158.528
C04287=1026.269,-15.813,-93.674,167.383,46.271,158.528
C04288=1026.275,-15.563,-93.688,167.386,46.269,158.528
C04289=1026.281,-15.314,-93.702,167.388,46.267,158.528
C04290=1026.287,-15.064,-93.716,167.391,46.264,158.527
C04291=1026.293,-14.815,-93.729,167.394,46.261,158.527
C04292=1026.299,-14.565,-93.743,167.396,46.259,158.527
C04293=1026.306,-14.315,-93.757,167.400,46.256,158.527
C04294=1026.311,-14.066,-93.771,167.402,46.254,158.527
C04295=1026.317,-13.816,-93.784,167.404,46.251,158.527
C04296=1026.323,-13.567,-93.798,167.408,46.248,158.526
C04297=1026.330,-13.318,-93.812,167.410,46.246,158.526
C04298=1026.336,-13.068,-93.826,167.412,46.243,158.526
C04299=1026.342,-12.819,-93.839,167.416,46.240,158.526
C04300=1026.348,-12.568,-93.854,167.418,46.238,158.526
C04301=1026.354,-12.319,-93.867,167.420,46.235,158.526
///RCONF 1,0,0,0,0,0,0,0,0,0,0,0,0,0,0,0,0,0,0,0,0,0,0,0
C04302=1026.360,-12.070,-93.881,167.423,46.232,158.525
C04303=1026.367,-11.820,-93.895,167.426,46.230,158.525
C04304=1026.372,-11.571,-93.909,167.429,46.227,158.525
C04305=1026.378,-11.321,-93.922,167.431,46.225,158.525
C04306=1026.384,-11.071,-93.936,167.434,46.222,158.525
C04307=1026.391,-10.822,-93.950,167.437,46.219,158.525
C04308=1026.397,-10.572,-93.965,167.439,46.217,158.524
C04309=1026.402,-10.323,-93.978,167.442,46.214,158.524
C04310=1026.409,-10.073,-93.992,167.445,46.212,158.524
C04311=1026.415,-9.823,-94.006,167.447,46.209,158.524
C04312=1026.421,-9.574,-94.020,167.450,46.207,158.524
C04313=1026.427,-9.325,-94.034,167.453,46.204,158.523
C04314=1026.434,-9.075,-94.047,167.455,46.201,158.523
C04315=1026.439,-8.826,-94.062,167.459,46.199,158.523
C04316=1026.446,-8.576,-94.076,167.461,46.196,158.523
C04317=1026.452,-8.326,-94.090,167.463,46.193,158.523
C04318=1026.458,-8.077,-94.103,167.466,46.190,158.523
C04319=1026.464,-7.828,-94.118,167.469,46.188,158.522
C04320=1026.470,-7.578,-94.131,167.471,46.185,158.522
C04321=1026.477,-7.328,-94.145,167.473,46.183,158.522
C04322=1026.482,-7.079,-94.160,167.477,46.180,158.522
C04323=1026.489,-6.829,-94.173,167.479,46.178,158.522
C04324=1026.495,-6.579,-94.187,167.481,46.175,158.521
C04325=1026.502,-6.330,-94.202,167.485,46.172,158.521
C04326=1026.507,-6.081,-94.216,167.487,46.170,158.521
C04327=1026.514,-5.832,-94.230,167.490,46.167,158.521
C04328=1026.520,-5.582,-94.244,167.493,46.164,158.521
C04329=1026.526,-5.332,-94.257,167.495,46.161,158.521
C04330=1026.532,-5.083,-94.272,167.498,46.159,158.520
C04331=1026.540,-4.800,-94.287,167.501,46.155,158.520
C04332=1026.546,-4.518,-94.303,167.504,46.152,158.520
C04333=1026.554,-4.236,-94.319,167.507,46.149,158.520
C04334=1026.560,-3.953,-94.335,167.509,46.147,158.520
C04335=1026.566,-3.704,-94.350,167.513,46.144,158.520
C04336=1026.572,-3.454,-94.364,167.515,46.142,158.519
C04337=1026.578,-3.205,-94.378,167.518,46.139,158.519
C04338=1026.585,-2.955,-94.392,167.520,46.137,158.519
C04339=1026.590,-2.706,-94.407,167.522,46.134,158.519
C04340=1026.597,-2.456,-94.422,167.526,46.132,158.519
C04341=1026.602,-2.207,-94.436,167.528,46.129,158.518
C04342=1026.609,-1.957,-94.451,167.531,46.127,158.518
C04343=1026.614,-1.707,-94.465,167.533,46.124,158.518
C04344=1026.620,-1.458,-94.480,167.537,46.122,158.518
C04345=1026.626,-1.209,-94.494,167.539,46.119,158.518
C04346=1026.632,-0.958,-94.508,167.541,46.116,158.518
C04347=1026.639,-0.710,-94.522,167.544,46.114,158.517
C04348=1026.645,-0.460,-94.537,167.547,46.111,158.517
C04349=1026.651,-0.211,-94.551,167.549,46.109,158.517
C04350=1026.657,0.039,-94.566,167.552,46.106,158.517
C04351=1026.663,0.288,-94.581,167.554,46.104,158.517
C04352=1026.669,0.538,-94.595,167.556,46.102,158.517
C04353=1026.675,0.787,-94.610,167.560,46.099,158.516
C04354=1026.681,1.037,-94.624,167.562,46.097,158.516
C04355=1026.687,1.287,-94.639,167.565,46.094,158.516
C04356=1026.693,1.536,-94.653,167.567,46.091,158.516
C04357=1026.699,1.786,-94.668,167.570,46.089,158.516
C04358=1026.705,2.035,-94.682,167.573,46.086,158.516
C04359=1026.712,2.285,-94.696,167.575,46.084,158.515
C04360=1026.718,2.534,-94.711,167.577,46.081,158.515
C04361=1026.724,2.783,-94.726,167.580,46.079,158.515
C04362=1026.730,3.034,-94.740,167.583,46.076,158.515
C04363=1026.736,3.283,-94.755,167.585,46.073,158.515
C04364=1026.742,3.532,-94.770,167.588,46.071,158.514
C04365=1026.748,3.781,-94.784,167.590,46.069,158.514
C04366=1026.754,4.031,-94.799,167.594,46.066,158.514
C04367=1026.761,4.281,-94.813,167.596,46.063,158.514
C04368=1026.766,4.530,-94.828,167.598,46.061,158.514
C04369=1026.773,4.780,-94.843,167.601,46.058,158.514
C04370=1026.779,5.029,-94.858,167.604,46.055,158.513
C04371=1026.785,5.279,-94.872,167.606,46.053,158.513
C04372=1026.791,5.529,-94.887,167.609,46.050,158.513
C04373=1026.798,5.777,-94.901,167.611,46.048,158.513
C04374=1026.804,6.027,-94.916,167.614,46.046,158.513
C04375=1026.810,6.277,-94.931,167.617,46.043,158.513
C04376=1026.816,6.526,-94.945,167.619,46.040,158.512
C04377=1026.822,6.776,-94.959,167.622,46.038,158.512
C04378=1026.829,7.025,-94.974,167.624,46.035,158.512
C04379=1026.834,7.274,-94.989,167.627,46.032,158.512
C04380=1026.841,7.524,-95.004,167.629,46.029,158.511
C04381=1026.847,7.774,-95.019,167.632,46.027,158.511
C04382=1026.853,8.023,-95.033,167.634,46.024,158.511
C04383=1026.859,8.272,-95.048,167.638,46.021,158.511
C04384=1026.866,8.522,-95.063,167.640,46.019,158.511
C04385=1026.871,8.771,-95.078,167.642,46.017,158.511
C04386=1026.877,9.021,-95.092,167.645,46.014,158.510
C04387=1026.884,9.271,-95.107,167.648,46.011,158.510
C04388=1026.890,9.521,-95.122,167.650,46.009,158.510
C04389=1026.896,9.769,-95.137,167.653,46.006,158.510
C04390=1026.902,10.019,-95.152,167.655,46.003,158.510
C04391=1026.909,10.269,-95.167,167.658,46.000,158.509
C04392=1026.915,10.518,-95.181,167.661,45.998,158.509
C04393=1026.922,10.767,-95.195,167.663,45.996,158.509
C04394=1026.928,11.017,-95.210,167.665,45.993,158.509
C04395=1026.935,11.301,-95.228,167.669,45.990,158.509
C04396=1026.942,11.586,-95.245,167.672,45.987,158.508
C04397=1026.949,11.869,-95.261,167.674,45.984,158.508
C04398=1026.956,12.154,-95.279,167.677,45.981,158.508
C04399=1026.962,12.403,-95.294,167.680,45.978,158.508
C04400=1026.969,12.653,-95.309,167.682,45.976,158.507
C04401=1026.975,12.903,-95.324,167.685,45.973,158.507
C04402=1026.981,13.152,-95.338,167.688,45.970,158.507
C04403=1026.988,13.401,-95.352,167.690,45.968,158.507
C04404=1026.994,13.651,-95.367,167.692,45.965,158.507
C04405=1027.000,13.901,-95.383,167.696,45.962,158.507
C04406=1027.006,14.150,-95.398,167.698,45.960,158.506
C04407=1027.012,14.399,-95.412,167.700,45.957,158.506
C04408=1027.019,14.649,-95.427,167.703,45.955,158.506
C04409=1027.025,14.898,-95.444,167.705,45.953,158.506
C04410=1027.031,15.148,-95.459,167.708,45.950,158.506
C04411=1027.037,15.398,-95.474,167.711,45.947,158.505
C04412=1027.043,15.647,-95.488,167.713,45.945,158.505
C04413=1027.049,15.897,-95.504,167.716,45.942,158.505
C04414=1027.055,16.146,-95.519,167.718,45.939,158.505
C04415=1027.062,16.395,-95.534,167.720,45.937,158.505
C04416=1027.068,16.645,-95.549,167.724,45.934,158.504
C04417=1027.073,16.894,-95.564,167.726,45.932,158.504
C04418=1027.080,17.144,-95.579,167.728,45.930,158.504
C04419=1027.086,17.393,-95.595,167.731,45.927,158.504
C04420=1027.093,17.642,-95.610,167.733,45.924,158.504
C04421=1027.098,17.892,-95.626,167.736,45.922,158.504
C04422=1027.105,18.141,-95.641,167.739,45.919,158.503
C04423=1027.111,18.390,-95.656,167.741,45.916,158.503
C04424=1027.117,18.640,-95.671,167.744,45.914,158.503
C04425=1027.123,18.890,-95.686,167.746,45.912,158.503
C04426=1027.130,19.139,-95.702,167.748,45.909,158.502
C04427=1027.136,19.389,-95.717,167.752,45.907,158.502
C04428=1027.142,19.638,-95.732,167.754,45.904,158.502
C04429=1027.148,19.888,-95.748,167.756,45.901,158.502
C04430=1027.154,20.137,-95.763,167.759,45.899,158.502
C04431=1027.160,20.387,-95.778,167.761,45.896,158.502
C04432=1027.166,20.636,-95.794,167.763,45.894,158.501
C04433=1027.173,20.885,-95.809,167.766,45.892,158.501
C04434=1027.178,21.135,-95.824,167.769,45.889,158.501
C04435=1027.185,21.384,-95.840,167.772,45.887,158.501
C04436=1027.191,21.634,-95.856,167.774,45.884,158.501
C04437=1027.197,21.883,-95.871,167.776,45.881,158.500
C04438=1027.203,22.132,-95.886,167.779,45.879,158.500
C04439=1027.209,22.382,-95.902,167.781,45.876,158.500
C04440=1027.216,22.631,-95.917,167.783,45.874,158.500
C04441=1027.221,22.881,-95.933,167.787,45.871,158.500
C04442=1027.228,23.130,-95.948,167.789,45.869,158.500
C04443=1027.234,23.380,-95.963,167.791,45.866,158.499
C04444=1027.240,23.629,-95.979,167.794,45.864,158.499
C04445=1027.247,23.879,-95.994,167.796,45.861,158.499
C04446=1027.253,24.128,-96.011,167.799,45.858,158.499
C04447=1027.259,24.378,-96.026,167.801,45.856,158.499
C04448=1027.265,24.627,-96.042,167.804,45.853,158.498
C04449=1027.271,24.877,-96.057,167.807,45.851,158.498
C04450=1027.278,25.126,-96.072,167.809,45.849,158.498
C04451=1027.284,25.376,-96.088,167.811,45.846,158.498
C04452=1027.290,25.625,-96.104,167.814,45.843,158.497
C04453=1027.296,25.875,-96.119,167.816,45.840,158.497
C04454=1027.302,26.123,-96.134,167.820,45.838,158.497
C04455=1027.308,26.373,-96.150,167.822,45.835,158.497
C04456=1027.314,26.622,-96.166,167.824,45.833,158.497
C04457=1027.320,26.872,-96.182,167.827,45.831,158.497
C04458=1027.327,27.121,-96.197,167.829,45.828,158.496
C04459=1027.333,27.407,-96.215,167.832,45.825,158.496
C04460=1027.342,27.693,-96.233,167.835,45.822,158.496
C04461=1027.348,27.978,-96.251,167.838,45.819,158.496
C04462=1027.355,28.265,-96.269,167.841,45.816,158.496
C04463=1027.362,28.514,-96.285,167.843,45.814,158.495
C04464=1027.368,28.763,-96.301,167.846,45.812,158.495
C04465=1027.374,29.012,-96.317,167.848,45.809,158.495
C04466=1027.380,29.262,-96.332,167.850,45.806,158.495
C04467=1027.386,29.511,-96.348,167.853,45.804,158.495
C04468=1027.393,29.760,-96.364,167.855,45.801,158.494
C04469=1027.398,30.010,-96.380,167.858,45.799,158.494
C04470=1027.404,30.260,-96.396,167.860,45.797,158.494
C04471=1027.411,30.509,-96.411,167.862,45.794,158.494
C04472=1027.417,30.758,-96.428,167.866,45.792,158.494
C04473=1027.422,31.008,-96.443,167.868,45.789,158.493
C04474=1027.429,31.257,-96.459,167.870,45.786,158.493
C04475=1027.435,31.506,-96.475,167.873,45.784,158.493
C04476=1027.441,31.756,-96.491,167.875,45.781,158.493
C04477=1027.447,32.005,-96.506,167.878,45.779,158.492
C04478=1027.453,32.255,-96.523,167.880,45.777,158.492
C04479=1027.459,32.504,-96.539,167.882,45.774,158.492
C04480=1027.466,32.753,-96.555,167.885,45.771,158.492
C04481=1027.472,33.003,-96.570,167.888,45.769,158.492
C04482=1027.478,33.252,-96.586,167.890,45.766,158.492
C04483=1027.484,33.501,-96.602,167.893,45.764,158.491
C04484=1027.490,33.751,-96.618,167.895,45.762,158.491
C04485=1027.497,34.001,-96.635,167.898,45.759,158.491
C04486=1027.503,34.250,-96.651,167.900,45.756,158.491
C04487=1027.509,34.500,-96.666,167.902,45.754,158.491
C04488=1027.515,34.749,-96.682,167.905,45.751,158.490
C04489=1027.522,34.998,-96.698,167.908,45.748,158.490
C04490=1027.528,35.248,-96.714,167.911,45.746,158.490
C04491=1027.534,35.497,-96.731,167.913,45.744,158.490
C04492=1027.540,35.746,-96.746,167.915,45.741,158.489
C04493=1027.546,35.995,-96.762,167.917,45.738,158.489
C04494=1027.552,36.245,-96.779,167.920,45.736,158.489
C04495=1027.559,36.495,-96.794,167.922,45.733,158.489
C04496=1027.565,36.744,-96.810,167.924,45.731,158.489
C04497=1027.571,36.994,-96.827,167.928,45.728,158.489
C04498=1027.577,37.243,-96.843,167.930,45.726,158.488
C04499=1027.583,37.492,-96.859,167.933,45.723,158.488
C04500=1027.589,37.742,-96.875,167.935,45.721,158.488
C04501=1027.596,37.991,-96.891,167.937,45.718,158.488
C04502=1027.602,38.240,-96.907,167.940,45.716,158.488
C04503=1027.608,38.490,-96.924,167.942,45.714,158.487
C04504=1027.614,38.740,-96.940,167.944,45.711,158.487
C04505=1027.620,38.989,-96.956,167.947,45.709,158.487
C04506=1027.626,39.238,-96.973,167.949,45.706,158.487
C04507=1027.632,39.488,-96.989,167.952,45.704,158.487
C04508=1027.638,39.737,-97.005,167.954,45.701,158.486
C04509=1027.644,39.986,-97.022,167.956,45.699,158.486
C04510=1027.651,40.236,-97.039,167.960,45.696,158.486
C04511=1027.657,40.485,-97.055,167.962,45.694,158.486
C04512=1027.663,40.734,-97.071,167.965,45.691,158.485
C04513=1027.669,40.983,-97.087,167.967,45.689,158.485
C04514=1027.675,41.233,-97.103,167.969,45.686,158.485
C04515=1027.682,41.483,-97.120,167.972,45.684,158.485
C04516=1027.688,41.732,-97.136,167.974,45.681,158.485
C04517=1027.694,41.982,-97.152,167.976,45.679,158.484
C04518=1027.700,42.231,-97.169,167.979,45.677,158.484
C04519=1027.706,42.480,-97.186,167.981,45.674,158.484
C04520=1027.712,42.730,-97.202,167.984,45.671,158.484
C04521=1027.718,42.979,-97.218,167.986,45.669,158.484
C04522=1027.724,43.228,-97.235,167.988,45.667,158.483
C04523=1027.731,43.514,-97.254,167.992,45.664,158.483
C04524=1027.738,43.800,-97.273,167.994,45.661,158.483
C04525=1027.745,44.085,-97.292,167.998,45.659,158.483
C04526=1027.751,44.371,-97.311,168.000,45.656,158.483
C04527=1027.758,44.620,-97.328,168.002,45.653,158.482
C04528=1027.764,44.869,-97.344,168.005,45.651,158.482
C04529=1027.770,45.119,-97.361,168.007,45.649,158.482
C04530=1027.775,45.368,-97.377,168.009,45.646,158.482
C04531=1027.782,45.617,-97.394,168.012,45.644,158.482
C04532=1027.788,45.867,-97.411,168.014,45.642,158.482
C04533=1027.794,46.117,-97.427,168.017,45.639,158.481
C04534=1027.800,46.365,-97.444,168.020,45.636,158.481
C04535=1027.805,46.615,-97.461,168.022,45.634,158.481
C04536=1027.812,46.865,-97.478,168.025,45.631,158.481
C04537=1027.818,47.114,-97.495,168.027,45.629,158.481
C04538=1027.824,47.363,-97.511,168.029,45.627,158.480
C04539=1027.830,47.612,-97.527,168.032,45.625,158.480
C04540=1027.836,47.862,-97.545,168.034,45.622,158.480
C04541=1027.842,48.111,-97.561,168.037,45.620,158.480
C04542=1027.849,48.360,-97.578,168.039,45.617,158.480
C04543=1027.854,48.610,-97.595,168.041,45.614,158.479
C04544=1027.861,48.860,-97.611,168.044,45.612,158.479
C04545=1027.867,49.109,-97.629,168.046,45.610,158.479
C04546=1027.873,49.358,-97.645,168.049,45.608,158.479
C04547=1027.879,49.607,-97.662,168.051,45.605,158.479
C04548=1027.885,49.857,-97.679,168.053,45.602,158.478
C04549=1027.891,50.106,-97.696,168.056,45.600,158.478
C04550=1027.897,50.355,-97.713,168.058,45.598,158.478
C04551=1027.903,50.605,-97.729,168.061,45.596,158.478
C04552=1027.910,50.854,-97.746,168.063,45.593,158.478
C04553=1027.916,51.103,-97.762,168.065,45.590,158.477
C04554=1027.922,51.353,-97.780,168.068,45.588,158.477
C04555=1027.928,51.602,-97.797,168.070,45.585,158.477
C04556=1027.934,51.851,-97.814,168.073,45.583,158.477
C04557=1027.940,52.101,-97.830,168.076,45.581,158.477
C04558=1027.946,52.350,-97.848,168.078,45.578,158.476
C04559=1027.952,52.600,-97.864,168.081,45.576,158.476
C04560=1027.959,52.849,-97.881,168.083,45.573,158.476
C04561=1027.965,53.098,-97.898,168.085,45.570,158.476
C04562=1027.971,53.347,-97.915,168.088,45.568,158.476
C04563=1027.977,53.597,-97.932,168.090,45.566,158.475
C04564=1027.983,53.846,-97.949,168.092,45.563,158.475
C04565=1027.989,54.095,-97.965,168.095,45.561,158.475
C04566=1027.996,54.345,-97.982,168.097,45.558,158.475
C04567=1028.001,54.595,-97.999,168.100,45.556,158.474
C04568=1028.008,54.844,-98.017,168.102,45.554,158.474
C04569=1028.014,55.093,-98.033,168.104,45.551,158.474
C04570=1028.020,55.342,-98.050,168.107,45.548,158.474
C04571=1028.026,55.592,-98.068,168.109,45.546,158.474
C04572=1028.032,55.841,-98.084,168.113,45.543,158.474
C04573=1028.039,56.091,-98.101,168.115,45.541,158.473
C04574=1028.045,56.340,-98.118,168.117,45.539,158.473
C04575=1028.051,56.589,-98.135,168.120,45.536,158.473
C04576=1028.057,56.838,-98.152,168.122,45.533,158.473
C04577=1028.063,57.088,-98.169,168.124,45.530,158.472
C04578=1028.070,57.337,-98.186,168.127,45.528,158.472
C04579=1028.075,57.587,-98.203,168.129,45.526,158.472
C04580=1028.082,57.836,-98.220,168.131,45.523,158.472
C04581=1028.089,58.085,-98.237,168.134,45.521,158.472
C04582=1028.094,58.334,-98.253,168.136,45.518,158.471
C04583=1028.101,58.584,-98.271,168.138,45.516,158.471
C04584=1028.107,58.833,-98.288,168.141,45.513,158.471
C04585=1028.113,59.083,-98.305,168.144,45.511,158.471
C04586=1028.120,59.332,-98.322,168.147,45.508,158.470
C04587=1028.127,59.618,-98.342,168.149,45.505,158.470
C04588=1028.134,59.902,-98.361,168.152,45.502,158.470
C04589=1028.141,60.188,-98.382,168.154,45.499,158.470
C04590=1028.148,60.473,-98.401,168.158,45.496,158.469
C04591=1028.155,60.722,-98.418,168.160,45.494,158.469
C04592=1028.161,60.971,-98.434,168.162,45.491,158.469
C04593=1028.167,61.221,-98.452,168.165,45.489,158.469
C04594=1028.173,61.470,-98.469,168.167,45.486,158.468
C04595=1028.180,61.720,-98.486,168.169,45.484,158.468
C04596=1028.185,61.969,-98.503,168.172,45.481,158.468
C04597=1028.192,62.218,-98.521,168.175,45.478,158.468
C04598=1028.198,62.467,-98.538,168.177,45.476,158.468
C04599=1028.205,62.717,-98.554,168.180,45.473,158.467
C04600=1028.211,62.966,-98.572,168.182,45.471,158.467
C04601=1028.217,63.216,-98.589,168.184,45.468,158.467
C04602=1028.224,63.465,-98.606,168.187,45.466,158.467
C04603=1028.230,63.714,-98.624,168.189,45.463,158.466
C04604=1028.237,63.964,-98.641,168.192,45.461,158.466
C04605=1028.242,64.213,-98.658,168.194,45.458,158.466
C04606=1028.249,64.463,-98.676,168.196,45.456,158.466
C04607=1028.254,64.712,-98.693,168.199,45.454,158.466
C04608=1028.260,64.961,-98.711,168.201,45.451,158.465
C04609=1028.267,65.210,-98.728,168.204,45.449,158.465
C04610=1028.273,65.460,-98.746,168.206,45.446,158.465
C04611=1028.279,65.709,-98.763,168.208,45.443,158.465
C04612=1028.285,65.958,-98.781,168.211,45.441,158.465
C04613=1028.291,66.207,-98.798,168.214,45.439,158.464
C04614=1028.297,66.457,-98.816,168.216,45.436,158.464
C04615=1028.303,66.706,-98.833,168.219,45.434,158.464
C04616=1028.310,66.955,-98.851,168.221,45.431,158.464
C04617=1028.315,67.204,-98.868,168.224,45.429,158.464
C04618=1028.322,67.454,-98.886,168.226,45.427,158.463
C04619=1028.328,67.704,-98.903,168.228,45.424,158.463
C04620=1028.334,67.953,-98.921,168.231,45.422,158.463
C04621=1028.341,68.202,-98.938,168.233,45.419,158.463
C04622=1028.346,68.451,-98.956,168.235,45.416,158.462
C04623=1028.353,68.700,-98.973,168.238,45.414,158.462
C04624=1028.359,68.950,-98.991,168.240,45.412,158.462
C04625=1028.365,69.199,-99.009,168.243,45.409,158.462
C04626=1028.371,69.449,-99.027,168.245,45.407,158.462
C04627=1028.377,69.698,-99.044,168.247,45.404,158.461
C04628=1028.383,69.947,-99.062,168.250,45.402,158.461
C04629=1028.389,70.196,-99.080,168.252,45.400,158.461
C04630=1028.395,70.446,-99.098,168.254,45.397,158.461
C04631=1028.402,70.695,-99.115,168.257,45.395,158.461
C04632=1028.408,70.944,-99.133,168.259,45.392,158.460
C04633=1028.414,71.194,-99.151,168.262,45.390,158.460
C04634=1028.419,71.443,-99.168,168.264,45.388,158.460
C04635=1028.426,71.692,-99.186,168.266,45.385,158.460
C04636=1028.432,71.941,-99.204,168.269,45.383,158.460
C04637=1028.438,72.190,-99.222,168.271,45.380,158.459
C04638=1028.444,72.440,-99.240,168.274,45.378,158.459
C04639=1028.450,72.689,-99.257,168.277,45.375,158.459
C04640=1028.456,72.939,-99.275,168.279,45.373,158.459
C04641=1028.463,73.188,-99.293,168.282,45.371,158.459
C04642=1028.468,73.437,-99.311,168.284,45.368,158.458
C04643=1028.475,73.687,-99.329,168.287,45.366,158.458
C04644=1028.481,73.936,-99.347,168.289,45.363,158.458
C04645=1028.487,74.184,-99.364,168.291,45.361,158.458
C04646=1028.493,74.434,-99.382,168.294,45.359,158.458
C04647=1028.499,74.684,-99.400,168.296,45.356,158.457
C04648=1028.505,74.933,-99.418,168.299,45.353,158.457
C04649=1028.511,75.182,-99.436,168.301,45.351,158.457
C04650=1028.518,75.432,-99.454,168.303,45.349,158.457
C04651=1028.525,75.716,-99.474,168.306,45.346,158.456
C04652=1028.532,76.001,-99.495,168.309,45.343,158.456
C04653=1028.540,76.287,-99.515,168.311,45.340,158.456
C04654=1028.546,76.571,-99.536,168.315,45.337,158.456
C04655=1028.552,76.821,-99.554,168.317,45.335,158.455
C04656=1028.558,77.071,-99.572,168.319,45.333,158.455
C04657=1028.564,77.319,-99.590,168.322,45.330,158.455
C04658=1028.570,77.569,-99.608,168.324,45.327,158.455
C04659=1028.576,77.819,-99.626,168.327,45.325,158.455
C04660=1028.582,78.067,-99.644,168.329,45.323,158.454
C04661=1028.588,78.317,-99.662,168.331,45.321,158.454
C04662=1028.595,78.566,-99.681,168.334,45.318,158.454
C04663=1028.601,78.816,-99.699,168.336,45.316,158.454
C04664=1028.606,79.065,-99.716,168.339,45.313,158.454
C04665=1028.613,79.314,-99.735,168.341,45.311,158.453
C04666=1028.618,79.564,-99.753,168.343,45.309,158.453
C04667=1028.624,79.812,-99.772,168.346,45.307,158.453
C04668=1028.630,80.062,-99.790,168.348,45.304,158.453
C04669=1028.637,80.311,-99.808,168.351,45.301,158.452
C04670=1028.642,80.560,-99.826,168.353,45.299,158.452
C04671=1028.649,80.809,-99.844,168.355,45.297,158.452
C04672=1028.655,81.059,-99.862,168.358,45.295,158.452
C04673=1028.661,81.308,-99.881,168.360,45.292,158.452
C04674=1028.667,81.557,-99.899,168.363,45.290,158.452
C04675=1028.673,81.806,-99.917,168.365,45.287,158.451
C04676=1028.680,82.056,-99.936,168.368,45.285,158.451
C04677=1028.686,82.305,-99.954,168.370,45.283,158.451
C04678=1028.691,82.554,-99.973,168.372,45.280,158.451
C04679=1028.697,82.804,-99.991,168.376,45.278,158.451
C04680=1028.703,83.053,-100.009,168.378,45.275,158.450
C04681=1028.709,83.303,-100.027,168.381,45.273,158.450
C04682=1028.715,83.551,-100.045,168.383,45.271,158.450
C04683=1028.721,83.801,-100.063,168.385,45.268,158.450
C04684=1028.728,84.050,-100.082,168.388,45.266,158.450
C04685=1028.734,84.299,-100.101,168.390,45.263,158.449
C04686=1028.740,84.549,-100.119,168.393,45.261,158.449
C04687=1028.746,84.797,-100.137,168.395,45.259,158.449
C04688=1028.753,85.046,-100.156,168.397,45.256,158.449
C04689=1028.758,85.296,-100.174,168.400,45.254,158.448
C04690=1028.764,85.545,-100.193,168.402,45.251,158.448
C04691=1028.770,85.795,-100.211,168.405,45.249,158.448
C04692=1028.776,86.044,-100.229,168.407,45.247,158.448
C04693=1028.783,86.293,-100.248,168.409,45.244,158.448
C04694=1028.789,86.543,-100.266,168.412,45.242,158.447
C04695=1028.795,86.792,-100.284,168.414,45.239,158.447
C04696=1028.802,87.041,-100.303,168.416,45.237,158.447
C04697=1028.808,87.290,-100.321,168.419,45.235,158.447
C04698=1028.813,87.539,-100.340,168.422,45.232,158.446
C04699=1028.819,87.788,-100.358,168.425,45.229,158.446
C04700=1028.825,88.038,-100.376,168.427,45.227,158.446
C04701=1028.832,88.287,-100.395,168.429,45.224,158.446
C04702=1028.838,88.536,-100.414,168.432,45.222,158.446
C04703=1028.845,88.785,-100.432,168.434,45.220,158.445
C04704=1028.851,89.035,-100.450,168.437,45.217,158.445
C04705=1028.857,89.284,-100.468,168.439,45.214,158.445
C04706=1028.863,89.533,-100.487,168.441,45.212,158.445
C04707=1028.869,89.782,-100.506,168.444,45.210,158.444
C04708=1028.875,90.032,-100.524,168.446,45.208,158.444
C04709=1028.881,90.281,-100.543,168.449,45.205,158.444
C04710=1028.887,90.530,-100.562,168.451,45.203,158.444
C04711=1028.893,90.780,-100.581,168.453,45.200,158.444
C04712=1028.899,91.029,-100.600,168.456,45.199,158.444
C04713=1028.906,91.278,-100.619,168.458,45.196,158.443
C04714=1028.911,91.527,-100.638,168.461,45.194,158.443
C04715=1028.918,91.812,-100.658,168.464,45.191,158.443
C04716=1028.925,92.097,-100.680,168.466,45.188,158.443
C04717=1028.931,92.383,-100.701,168.470,45.185,158.442
C04718=1028.939,92.667,-100.723,168.472,45.183,158.442
C04719=1028.945,92.917,-100.742,168.475,45.181,158.442
C04720=1028.951,93.166,-100.761,168.477,45.178,158.442
C04721=1028.957,93.415,-100.780,168.479,45.175,158.441
C04722=1028.963,93.664,-100.798,168.482,45.174,158.441
C04723=1028.969,93.913,-100.817,168.484,45.171,158.441
C04724=1028.975,94.162,-100.836,168.487,45.169,158.441
C04725=1028.981,94.412,-100.855,168.490,45.166,158.441
C04726=1028.987,94.661,-100.874,168.492,45.164,158.441
C04727=1028.993,94.910,-100.893,168.495,45.161,158.440
C04728=1029.000,95.159,-100.911,168.497,45.159,158.440
C04729=1029.005,95.409,-100.931,168.500,45.157,158.440
C04730=1029.012,95.658,-100.949,168.502,45.154,158.440
C04731=1029.017,95.907,-100.968,168.505,45.152,158.440
C04732=1029.024,96.156,-100.987,168.507,45.149,158.439
C04733=1029.030,96.406,-101.006,168.509,45.147,158.439
C04734=1029.036,96.655,-101.025,168.512,45.145,158.439
C04735=1029.042,96.904,-101.044,168.514,45.143,158.439
C04736=1029.048,97.153,-101.063,168.517,45.140,158.438
C04737=1029.054,97.403,-101.082,168.519,45.137,158.438
C04738=1029.060,97.652,-101.101,168.521,45.135,158.438
C04739=1029.067,97.901,-101.119,168.524,45.133,158.438
C04740=1029.072,98.151,-101.139,168.526,45.131,158.438
C04741=1029.079,98.400,-101.157,168.530,45.128,158.437
C04742=1029.085,98.649,-101.176,168.532,45.125,158.437
C04743=1029.091,98.898,-101.195,168.534,45.123,158.437
C04744=1029.097,99.147,-101.214,168.537,45.121,158.437
C04745=1029.103,99.396,-101.234,168.539,45.119,158.437
C04746=1029.110,99.645,-101.252,168.542,45.116,158.436
C04747=1029.115,99.864,-101.269,168.544,45.114,158.436
C04748=1029.119,100.083,-101.286,168.546,45.112,158.436
C04749=1029.125,100.303,-101.303,168.548,45.110,158.436
C04750=1029.130,100.522,-101.320,168.551,45.108,158.436
C04751=1029.136,100.742,-101.336,168.552,45.106,158.435
C04752=1029.141,100.961,-101.353,168.555,45.104,158.435
C04753=1029.146,101.179,-101.371,168.557,45.102,158.435
C04754=1029.152,101.399,-101.387,168.558,45.100,158.435
C04755=1029.157,101.649,-101.407,168.561,45.098,158.435
C04756=1029.163,101.898,-101.426,168.565,45.095,158.435
C04757=1029.170,102.146,-101.445,168.567,45.093,158.434
C04758=1029.176,102.396,-101.465,168.569,45.091,158.434
C04759=1029.181,102.645,-101.484,168.572,45.088,158.434
C04760=1029.188,102.894,-101.502,168.574,45.086,158.434
C04761=1029.194,103.143,-101.522,168.577,45.083,158.434
C04762=1029.199,103.393,-101.542,168.579,45.081,158.433
C04763=1029.205,103.642,-101.561,168.581,45.079,158.433
C04764=1029.212,103.891,-101.580,168.584,45.077,158.433
C04765=1029.217,104.140,-101.599,168.586,45.074,158.433
C04766=1029.223,104.390,-101.619,168.589,45.072,158.433
C04767=1029.230,104.638,-101.638,168.591,45.070,158.432
C04768=1029.236,104.887,-101.657,168.594,45.068,158.432
C04769=1029.241,105.137,-101.677,168.596,45.065,158.432
C04770=1029.247,105.386,-101.697,168.599,45.063,158.432
C04771=1029.254,105.636,-101.716,168.601,45.060,158.432
C04772=1029.260,105.885,-101.735,168.604,45.058,158.431
C04773=1029.266,106.134,-101.755,168.607,45.056,158.431
C04774=1029.272,106.383,-101.773,168.609,45.053,158.431
C04775=1029.278,106.632,-101.793,168.612,45.051,158.431
C04776=1029.284,106.881,-101.813,168.614,45.048,158.431
C04777=1029.290,107.131,-101.832,168.617,45.046,158.430
C04778=1029.296,107.379,-101.851,168.619,45.044,158.430
C04779=1029.305,107.725,-101.878,168.622,45.041,158.430
C04780=1029.313,108.069,-101.906,168.626,45.037,158.430
C04781=1029.322,108.415,-101.932,168.630,45.034,158.429
C04782=1029.330,108.759,-101.959,168.633,45.031,158.429
C04783=1029.336,109.008,-101.979,168.635,45.029,158.429
C04784=1029.342,109.258,-101.998,168.637,45.026,158.429
C04785=1029.348,109.506,-102.017,168.641,45.024,158.428
C04786=1029.355,109.756,-102.037,168.643,45.021,158.428
C04787=1029.361,110.005,-102.057,168.646,45.019,158.428
C04788=1029.366,110.255,-102.076,168.648,45.017,158.428
C04789=1029.372,110.503,-102.096,168.651,45.014,158.428
C04790=1029.378,110.753,-102.115,168.653,45.012,158.427
C04791=1029.385,111.001,-102.135,168.656,45.010,158.427
C04792=1029.391,111.251,-102.155,168.658,45.007,158.427
C04793=1029.397,111.500,-102.174,168.661,45.005,158.427
C04794=1029.403,111.749,-102.194,168.663,45.003,158.427
C04795=1029.409,111.999,-102.213,168.666,45.001,158.426
C04796=1029.415,112.247,-102.233,168.669,44.998,158.426
C04797=1029.421,112.496,-102.253,168.671,44.996,158.426
C04798=1029.427,112.746,-102.273,168.674,44.993,158.426
C04799=1029.433,112.995,-102.293,168.676,44.991,158.426
C04800=1029.439,113.244,-102.313,168.678,44.989,158.425
C04801=1029.445,113.493,-102.332,168.681,44.987,158.425
C04802=1029.451,113.742,-102.352,168.684,44.985,158.425
C04803=1029.457,113.992,-102.373,168.686,44.982,158.425
C04804=1029.462,114.241,-102.392,168.688,44.980,158.425
C04805=1029.468,114.490,-102.412,168.691,44.978,158.425
C04806=1029.474,114.739,-102.432,168.693,44.976,158.424
C04807=1029.480,114.988,-102.452,168.696,44.974,158.424
C04808=1029.486,115.237,-102.472,168.698,44.972,158.424
C04809=1029.492,115.487,-102.492,168.702,44.969,158.424
C04810=1029.498,115.736,-102.512,168.704,44.967,158.424
C04811=1029.504,115.985,-102.532,168.707,44.964,158.423
C04812=1029.510,116.234,-102.552,168.709,44.962,158.423
C04813=1029.516,116.482,-102.572,168.712,44.960,158.423
C04814=1029.521,116.733,-102.592,168.714,44.958,158.423
C04815=1029.527,116.982,-102.612,168.717,44.956,158.423
C04816=1029.533,117.230,-102.632,168.719,44.954,158.423
C04817=1029.539,117.479,-102.652,168.721,44.951,158.422
C04818=1029.545,117.728,-102.672,168.724,44.949,158.422
C04819=1029.551,117.978,-102.693,168.727,44.947,158.422
C04820=1029.557,118.227,-102.713,168.729,44.944,158.422
C04821=1029.563,118.476,-102.732,168.732,44.942,158.422
C04822=1029.569,118.725,-102.752,168.735,44.940,158.421
C04823=1029.575,118.975,-102.773,168.737,44.938,158.421
C04824=1029.581,119.224,-102.793,168.740,44.936,158.421
C04825=1029.587,119.472,-102.813,168.742,44.933,158.421
C04826=1029.593,119.721,-102.833,168.745,44.931,158.421
C04827=1029.599,119.971,-102.853,168.747,44.929,158.420
C04828=1029.605,120.220,-102.873,168.750,44.927,158.420
C04829=1029.610,120.469,-102.894,168.752,44.925,158.420
C04830=1029.617,120.718,-102.914,168.756,44.922,158.420
C04831=1029.623,120.967,-102.934,168.758,44.920,158.420
C04832=1029.629,121.216,-102.954,168.760,44.917,158.420
C04833=1029.635,121.465,-102.974,168.763,44.915,158.419
C04834=1029.641,121.714,-102.995,168.765,44.913,158.419
C04835=1029.647,121.964,-103.014,168.768,44.911,158.419
C04836=1029.653,122.213,-103.034,168.770,44.909,158.419
C04837=1029.659,122.462,-103.054,168.773,44.906,158.419
C04838=1029.664,122.711,-103.075,168.776,44.904,158.419
C04839=1029.670,122.960,-103.095,168.779,44.901,158.418
C04840=1029.677,123.210,-103.115,168.781,44.899,158.418
C04841=1029.683,123.458,-103.136,168.784,44.897,158.418
C04842=1029.689,123.707,-103.156,168.786,44.895,158.418
C04843=1029.696,123.993,-103.179,168.789,44.892,158.417
C04844=1029.702,124.277,-103.202,168.792,44.890,158.417
C04845=1029.710,124.562,-103.225,168.795,44.887,158.417
C04846=1029.717,124.847,-103.249,168.799,44.884,158.417
C04847=1029.723,125.096,-103.268,168.801,44.882,158.417
C04848=1029.729,125.345,-103.289,168.803,44.880,158.416
C04849=1029.735,125.594,-103.310,168.806,44.878,158.416
C04850=1029.741,125.843,-103.330,168.808,44.875,158.416
C04851=1029.747,126.092,-103.350,168.811,44.873,158.416
C04852=1029.753,126.341,-103.370,168.814,44.870,158.416
C04853=1029.759,126.591,-103.391,168.817,44.868,158.416
C04854=1029.765,126.840,-103.411,168.819,44.866,158.415
C04855=1029.772,127.089,-103.432,168.822,44.864,158.415
C04856=1029.778,127.338,-103.451,168.824,44.862,158.415
C04857=1029.784,127.587,-103.471,168.828,44.859,158.415
C04858=1029.790,127.836,-103.493,168.830,44.857,158.415
C04859=1029.796,128.085,-103.513,168.832,44.854,158.414
C04860=1029.802,128.334,-103.533,168.835,44.852,158.414
C04861=1029.808,128.583,-103.553,168.837,44.850,158.414
C04862=1029.814,128.833,-103.574,168.841,44.848,158.414
C04863=1029.820,129.082,-103.594,168.843,44.845,158.414
C04864=1029.827,129.330,-103.615,168.846,44.843,158.413
C04865=1029.833,129.580,-103.635,168.848,44.840,158.413
C04866=1029.838,129.829,-103.656,168.851,44.838,158.413
C04867=1029.845,130.078,-103.676,168.854,44.836,158.413
C04868=1029.851,130.326,-103.697,168.856,44.834,158.413
C04869=1029.857,130.576,-103.718,168.859,44.832,158.412
C04870=1029.863,130.825,-103.738,168.861,44.829,158.412
C04871=1029.869,131.075,-103.759,168.864,44.827,158.412
C04872=1029.875,131.323,-103.779,168.867,44.825,158.412
C04873=1029.881,131.573,-103.800,168.870,44.822,158.412
C04874=1029.888,131.821,-103.821,168.872,44.820,158.412
C04875=1029.893,132.070,-103.841,168.875,44.818,158.411
C04876=1029.899,132.320,-103.862,168.877,44.816,158.411
C04877=1029.905,132.568,-103.883,168.880,44.814,158.411
C04878=1029.911,132.818,-103.904,168.883,44.812,158.411
C04879=1029.917,133.066,-103.925,168.886,44.810,158.411
C04880=1029.923,133.316,-103.945,168.888,44.807,158.411
C04881=1029.929,133.565,-103.965,168.891,44.805,158.410
C04882=1029.935,133.814,-103.987,168.893,44.803,158.410
C04883=1029.940,134.063,-104.008,168.897,44.800,158.410
C04884=1029.947,134.312,-104.029,168.899,44.798,158.410
C04885=1029.953,134.561,-104.049,168.902,44.796,158.410
C04886=1029.959,134.810,-104.070,168.904,44.794,158.409
C04887=1029.965,135.059,-104.091,168.907,44.792,158.409
C04888=1029.972,135.308,-104.112,168.909,44.790,158.409
C04889=1029.977,135.557,-104.132,168.913,44.788,158.409
C04890=1029.983,135.806,-104.154,168.915,44.785,158.409
C04891=1029.989,136.055,-104.174,168.918,44.783,158.409
C04892=1029.995,136.305,-104.196,168.920,44.781,158.409
C04893=1030.001,136.553,-104.216,168.924,44.778,158.408
C04894=1030.007,136.803,-104.237,168.926,44.777,158.408
C04895=1030.013,137.052,-104.258,168.929,44.775,158.408
C04896=1030.019,137.301,-104.279,168.931,44.772,158.408
C04897=1030.025,137.550,-104.300,168.934,44.770,158.408
C04898=1030.031,137.799,-104.321,168.937,44.768,158.408
C04899=1030.038,138.048,-104.342,168.940,44.766,158.407
C04900=1030.043,138.297,-104.363,168.942,44.763,158.407
C04901=1030.049,138.546,-104.384,168.945,44.761,158.407
C04902=1030.054,138.795,-104.405,168.948,44.759,158.407
C04903=1030.061,139.044,-104.426,168.951,44.757,158.407
C04904=1030.068,139.293,-104.447,168.953,44.755,158.406
C04905=1030.073,139.542,-104.468,168.956,44.753,158.406
C04906=1030.079,139.792,-104.490,168.958,44.751,158.406
C04907=1030.086,140.076,-104.514,168.962,44.748,158.406
C04908=1030.093,140.360,-104.538,168.965,44.746,158.406
C04909=1030.099,140.646,-104.562,168.967,44.743,158.406
C04910=1030.106,140.930,-104.586,168.971,44.741,158.406
C04911=1030.112,141.179,-104.608,168.974,44.739,158.405
C04912=1030.118,141.428,-104.629,168.976,44.736,158.405
C04913=1030.124,141.678,-104.650,168.980,44.734,158.405
C04914=1030.130,141.927,-104.671,168.982,44.732,158.405
C04915=1030.136,142.175,-104.692,168.985,44.730,158.405
C04916=1030.142,142.424,-104.714,168.987,44.728,158.404
C04917=1030.147,142.673,-104.735,168.991,44.726,158.404
C04918=1030.154,142.923,-104.756,168.993,44.724,158.404
C04919=1030.160,143.172,-104.778,168.996,44.722,158.404
C04920=1030.166,143.420,-104.799,168.998,44.720,158.404
C04921=1030.172,143.669,-104.820,169.002,44.717,158.404
C04922=1030.178,143.919,-104.842,169.004,44.715,158.404
C04923=1030.184,144.168,-104.862,169.007,44.713,158.403
C04924=1030.190,144.417,-104.884,169.009,44.711,158.403
C04925=1030.196,144.666,-104.906,169.013,44.708,158.403
C04926=1030.202,144.915,-104.927,169.015,44.706,158.403
C04927=1030.208,145.163,-104.948,169.018,44.704,158.403
C04928=1030.215,145.413,-104.970,169.020,44.702,158.403
C04929=1030.220,145.661,-104.991,169.024,44.700,158.403
C04930=1030.226,145.911,-105.012,169.026,44.698,158.402
C04931=1030.232,146.160,-105.033,169.029,44.696,158.402
C04932=1030.238,146.409,-105.055,169.032,44.694,158.402
C04933=1030.244,146.658,-105.076,169.035,44.692,158.402
C04934=1030.250,146.907,-105.098,169.037,44.690,158.402
C04935=1030.256,147.156,-105.119,169.040,44.687,158.401
C04936=1030.262,147.405,-105.141,169.043,44.685,158.401
C04937=1030.268,147.654,-105.163,169.046,44.683,158.401
C04938=1030.274,147.903,-105.184,169.048,44.681,158.401
C04939=1030.280,148.152,-105.205,169.051,44.679,158.401
C04940=1030.286,148.401,-105.227,169.055,44.677,158.401
C04941=1030.292,148.650,-105.249,169.057,44.675,158.401
C04942=1030.298,148.899,-105.270,169.060,44.673,158.401
C04943=1030.304,149.148,-105.292,169.062,44.671,158.400
C04944=1030.310,149.397,-105.313,169.066,44.668,158.400
C04945=1030.316,149.645,-105.335,169.068,44.666,158.400
C04946=1030.321,149.894,-105.357,169.071,44.665,158.400
C04947=1030.327,150.144,-105.379,169.074,44.662,158.400
C04948=1030.334,150.393,-105.401,169.077,44.660,158.400
C04949=1030.339,150.641,-105.422,169.079,44.658,158.400
C04950=1030.345,150.891,-105.444,169.082,44.657,158.399
C04951=1030.351,151.140,-105.465,169.086,44.654,158.399
C04952=1030.358,151.389,-105.487,169.088,44.652,158.399
C04953=1030.363,151.637,-105.509,169.091,44.650,158.399
C04954=1030.369,151.886,-105.531,169.094,44.648,158.399
C04955=1030.375,152.136,-105.553,169.097,44.646,158.399
C04956=1030.381,152.385,-105.574,169.099,44.644,158.399
C04957=1030.387,152.634,-105.596,169.103,44.642,158.398
C04958=1030.393,152.882,-105.618,169.105,44.640,158.398
C04959=1030.399,153.131,-105.640,169.108,44.638,158.398
C04960=1030.406,153.380,-105.661,169.111,44.636,158.398
C04961=1030.411,153.630,-105.683,169.114,44.634,158.398
C04962=1030.417,153.879,-105.705,169.116,44.631,158.398
C04963=1030.423,154.127,-105.727,169.119,44.629,158.398
C04964=1030.429,154.376,-105.749,169.123,44.627,158.397
C04965=1030.435,154.626,-105.771,169.125,44.625,158.397
C04966=1030.441,154.874,-105.793,169.128,44.623,158.397
C04967=1030.447,155.123,-105.815,169.131,44.621,158.397
C04968=1030.453,155.372,-105.836,169.134,44.619,158.397
C04969=1030.459,155.621,-105.859,169.136,44.617,158.397
C04970=1030.465,155.870,-105.881,169.140,44.615,158.397
C04971=1030.472,156.154,-105.906,169.143,44.613,158.397
C04972=1030.479,156.439,-105.931,169.146,44.611,158.396
C04973=1030.485,156.723,-105.956,169.149,44.608,158.396
C04974=1030.492,157.008,-105.981,169.153,44.606,158.396
C04975=1030.498,157.257,-106.003,169.156,44.604,158.396
C04976=1030.504,157.506,-106.026,169.158,44.602,158.396
C04977=1030.510,157.755,-106.048,169.162,44.600,158.396
C04978=1030.516,158.004,-106.070,169.164,44.598,158.396
C04979=1030.522,158.252,-106.091,169.168,44.596,158.396
C04980=1030.528,158.501,-106.114,169.170,44.594,158.395
C04981=1030.534,158.751,-106.136,169.173,44.592,158.395
C04982=1030.540,158.999,-106.158,169.177,44.590,158.395
C04983=1030.546,159.249,-106.180,169.179,44.588,158.395
C04984=1030.552,159.497,-106.202,169.182,44.586,158.395
C04985=1030.558,159.746,-106.224,169.185,44.584,158.395
C04986=1030.564,159.995,-106.247,169.188,44.582,158.395
C04987=1030.569,160.245,-106.269,169.190,44.580,158.395
C04988=1030.575,160.493,-106.292,169.194,44.578,158.394
C04989=1030.581,160.742,-106.314,169.197,44.577,158.394
C04990=1030.586,160.991,-106.336,169.199,44.575,158.394
C04991=1030.592,161.240,-106.359,169.202,44.573,158.394
C04992=1030.598,161.489,-106.382,169.206,44.571,158.394
C04993=1030.604,161.738,-106.404,169.208,44.569,158.394
C04994=1030.610,161.987,-106.427,169.211,44.567,158.394
C04995=1030.615,162.236,-106.450,169.215,44.565,158.394
C04996=1030.621,162.484,-106.472,169.217,44.563,158.394
C04997=1030.627,162.733,-106.494,169.220,44.561,158.394
C04998=1030.633,162.982,-106.517,169.223,44.559,158.393
C04999=1030.638,163.231,-106.540,169.226,44.558,158.393
C05000=1030.645,163.480,-106.562,169.229,44.556,158.393
C05001=1030.650,163.729,-106.585,169.232,44.554,158.393
C05002=1030.656,163.978,-106.608,169.235,44.552,158.393
C05003=1030.662,164.227,-106.630,169.237,44.550,158.393
C05004=1030.668,164.476,-106.653,169.241,44.549,158.393
C05005=1030.673,164.725,-106.675,169.244,44.547,158.393
C05006=1030.679,164.974,-106.698,169.246,44.545,158.393
C05007=1030.685,165.223,-106.721,169.250,44.543,158.393
C05008=1030.691,165.472,-106.743,169.252,44.541,158.392
C05009=1030.697,165.720,-106.766,169.256,44.539,158.393
C05010=1030.703,165.969,-106.789,169.259,44.537,158.392
C05011=1030.708,166.219,-106.811,169.261,44.535,158.392
C05012=1030.715,166.467,-106.834,169.265,44.533,158.392
C05013=1030.721,166.716,-106.857,169.268,44.532,158.392
C05014=1030.726,166.965,-106.879,169.270,44.530,158.392
C05015=1030.731,167.213,-106.902,169.274,44.528,158.392
C05016=1030.738,167.463,-106.925,169.276,44.526,158.392
C05017=1030.744,167.712,-106.948,169.280,44.524,158.392
C05018=1030.750,167.960,-106.971,169.283,44.523,158.392
C05019=1030.755,168.210,-106.993,169.285,44.521,158.392
C05020=1030.762,168.459,-107.015,169.289,44.519,158.391
C05021=1030.768,168.707,-107.038,169.292,44.517,158.391
C05022=1030.773,168.956,-107.061,169.295,44.515,158.391
C05023=1030.779,169.205,-107.084,169.298,44.513,158.391
C05024=1030.785,169.454,-107.107,169.301,44.511,158.391
C05025=1030.791,169.703,-107.130,169.304,44.509,158.391
C05026=1030.797,169.952,-107.153,169.307,44.507,158.391
C05027=1030.803,170.201,-107.175,169.311,44.506,158.391
C05028=1030.809,170.449,-107.198,169.313,44.504,158.391
C05029=1030.815,170.698,-107.221,169.317,44.502,158.391
C05030=1030.821,170.947,-107.244,169.319,44.500,158.391
C05031=1030.826,171.196,-107.267,169.323,44.498,158.390
C05032=1030.832,171.445,-107.290,169.326,44.496,158.390
C05033=1030.839,171.694,-107.312,169.328,44.495,158.390
C05034=1030.845,171.943,-107.335,169.332,44.492,158.390
C05035=1030.851,172.226,-107.361,169.335,44.490,158.390
C05036=1030.858,172.510,-107.387,169.339,44.488,158.390
C05037=1030.865,172.795,-107.414,169.343,44.486,158.390
C05038=1030.872,173.078,-107.440,169.346,44.484,158.390
C05039=1030.878,173.327,-107.463,169.349,44.482,158.390
C05040=1030.884,173.576,-107.486,169.352,44.480,158.390
C05041=1030.890,173.825,-107.509,169.355,44.479,158.390
C05042=1030.896,174.074,-107.532,169.359,44.476,158.390
C05043=1030.902,174.323,-107.555,169.361,44.475,158.389
C05044=1030.908,174.572,-107.578,169.365,44.473,158.389
C05045=1030.914,174.820,-107.601,169.368,44.471,158.389
C05046=1030.920,175.069,-107.624,169.371,44.469,158.389
C05047=1030.927,175.319,-107.647,169.374,44.467,158.389
C05048=1030.932,175.568,-107.670,169.378,44.466,158.389
C05049=1030.938,175.816,-107.693,169.380,44.464,158.389
C05050=1030.945,176.064,-107.716,169.384,44.462,158.389
C05051=1030.951,176.313,-107.739,169.386,44.460,158.389
C05052=1030.957,176.563,-107.762,169.390,44.458,158.389
C05053=1030.963,176.812,-107.785,169.393,44.456,158.389
C05054=1030.968,177.061,-107.808,169.396,44.454,158.389
C05055=1030.975,177.309,-107.831,169.399,44.452,158.388
C05056=1030.981,177.558,-107.855,169.403,44.451,158.388
C05057=1030.987,177.807,-107.878,169.405,44.449,158.388
C05058=1030.993,178.055,-107.901,169.409,44.447,158.388
C05059=1030.999,178.304,-107.924,169.412,44.445,158.388
C05060=1031.006,178.554,-107.947,169.415,44.443,158.388
C05061=1031.012,178.803,-107.970,169.419,44.441,158.388
C05062=1031.018,179.051,-107.993,169.421,44.439,158.388
C05063=1031.024,179.300,-108.017,169.425,44.437,158.388
C05064=1031.030,179.549,-108.040,169.428,44.436,158.388
C05065=1031.036,179.798,-108.063,169.431,44.434,158.388
C05066=1031.042,180.046,-108.086,169.434,44.432,158.388
C05067=1031.049,180.296,-108.109,169.438,44.430,158.388
C05068=1031.055,180.544,-108.133,169.441,44.428,158.387
C05069=1031.060,180.793,-108.156,169.444,44.426,158.387
C05070=1031.067,181.042,-108.180,169.447,44.424,158.387
C05071=1031.074,181.291,-108.202,169.450,44.423,158.387
C05072=1031.080,181.540,-108.225,169.454,44.421,158.387
C05073=1031.086,181.788,-108.249,169.457,44.419,158.387
C05074=1031.092,182.037,-108.272,169.460,44.417,158.387
C05075=1031.098,182.286,-108.296,169.464,44.415,158.387
C05076=1031.104,182.535,-108.319,169.466,44.413,158.387
C05077=1031.111,182.783,-108.342,169.470,44.412,158.387
C05078=1031.117,183.033,-108.365,169.474,44.410,158.387
C05079=1031.122,183.281,-108.390,169.477,44.409,158.387
C05080=1031.128,183.530,-108.413,169.480,44.406,158.387
C05081=1031.134,183.780,-108.437,169.483,44.405,158.387
C05082=1031.140,184.028,-108.461,169.487,44.403,158.387
C05083=1031.145,184.276,-108.485,169.489,44.402,158.387
C05084=1031.152,184.526,-108.508,169.493,44.400,158.387
C05085=1031.158,184.774,-108.532,169.496,44.398,158.386
C05086=1031.163,185.023,-108.556,169.500,44.397,158.387
C05087=1031.169,185.271,-108.580,169.502,44.395,158.386
C05088=1031.175,185.521,-108.604,169.506,44.394,158.386
C05089=1031.181,185.769,-108.628,169.509,44.392,158.386
C05090=1031.186,186.018,-108.652,169.512,44.390,158.386
C05091=1031.193,186.267,-108.676,169.516,44.389,158.386
C05092=1031.199,186.515,-108.699,169.519,44.388,158.386
C05093=1031.204,186.765,-108.723,169.523,44.385,158.386
C05094=1031.210,187.013,-108.747,169.525,44.384,158.386
C05095=1031.216,187.262,-108.771,169.529,44.383,158.386
C05096=1031.222,187.511,-108.795,169.532,44.381,158.386
C05097=1031.228,187.759,-108.820,169.536,44.379,158.386
C05098=1031.234,188.008,-108.843,169.539,44.378,158.386
C05099=1031.240,188.292,-108.870,169.543,44.376,158.386
C05100=1031.247,188.575,-108.898,169.547,44.374,158.386
C05101=1031.254,188.859,-108.925,169.550,44.372,158.386
C05102=1031.261,189.143,-108.952,169.554,44.370,158.386
C05103=1031.267,189.392,-108.977,169.558,44.369,158.386
C05104=1031.273,189.640,-109.000,169.561,44.367,158.386
C05105=1031.279,189.890,-109.025,169.564,44.365,158.386
C05106=1031.285,190.138,-109.049,169.567,44.364,158.386
C05107=1031.291,190.387,-109.073,169.571,44.363,158.386
C05108=1031.297,190.635,-109.097,169.574,44.360,158.386
C05109=1031.303,190.884,-109.121,169.577,44.359,158.386
C05110=1031.308,191.133,-109.145,169.581,44.358,158.386
C05111=1031.315,191.381,-109.169,169.585,44.356,158.386
C05112=1031.320,191.631,-109.193,169.587,44.354,158.386
C05113=1031.326,191.879,-109.217,169.591,44.353,158.386
C05114=1031.332,192.128,-109.242,169.595,44.351,158.386
C05115=1031.338,192.376,-109.265,169.598,44.349,158.386
C05116=1031.344,192.626,-109.290,169.601,44.348,158.386
C05117=1031.351,192.875,-109.314,169.605,44.347,158.386
C05118=1031.356,193.123,-109.338,169.608,44.345,158.386
C05119=1031.363,193.372,-109.362,169.612,44.343,158.386
C05120=1031.368,193.621,-109.387,169.615,44.342,158.386
C05121=1031.375,193.869,-109.411,169.618,44.340,158.386
C05122=1031.380,194.118,-109.436,169.622,44.338,158.386
C05123=1031.387,194.367,-109.460,169.626,44.337,158.386
C05124=1031.393,194.615,-109.483,169.629,44.336,158.386
C05125=1031.399,194.864,-109.508,169.632,44.334,158.386
C05126=1031.406,195.113,-109.532,169.636,44.332,158.386
C05127=1031.411,195.362,-109.556,169.639,44.331,158.386
C05128=1031.418,195.610,-109.581,169.643,44.329,158.386
C05129=1031.423,195.859,-109.605,169.646,44.327,158.386
C05130=1031.430,196.108,-109.629,169.650,44.326,158.386
C05131=1031.436,196.357,-109.654,169.653,44.325,158.386
C05132=1031.442,196.605,-109.677,169.657,44.323,158.386
C05133=1031.448,196.854,-109.703,169.660,44.321,158.386
C05134=1031.455,197.103,-109.727,169.663,44.320,158.386
C05135=1031.460,197.352,-109.751,169.667,44.318,158.386
C05136=1031.467,197.601,-109.775,169.671,44.317,158.386
C05137=1031.473,197.849,-109.800,169.674,44.315,158.386
C05138=1031.479,198.098,-109.824,169.677,44.313,158.386
C05139=1031.485,198.347,-109.849,169.681,44.312,158.386
C05140=1031.492,198.595,-109.873,169.685,44.311,158.386
C05141=1031.497,198.844,-109.898,169.688,44.309,158.386
C05142=1031.504,199.093,-109.922,169.691,44.307,158.386
C05143=1031.510,199.341,-109.947,169.695,44.306,158.386
C05144=1031.516,199.590,-109.971,169.699,44.304,158.386
C05145=1031.522,199.839,-109.995,169.702,44.303,158.386
C05146=1031.529,200.087,-110.020,169.706,44.301,158.386
C05147=1031.535,200.337,-110.045,169.709,44.299,158.386
C05148=1031.540,200.585,-110.069,169.713,44.298,158.386
C05149=1031.547,200.834,-110.094,169.717,44.297,158.386
C05150=1031.553,201.083,-110.118,169.720,44.295,158.386
C05151=1031.559,201.332,-110.144,169.723,44.294,158.386
C05152=1031.564,201.579,-110.169,169.727,44.292,158.386
C05153=1031.570,201.829,-110.193,169.731,44.291,158.386
C05154=1031.577,202.077,-110.219,169.735,44.289,158.386
C05155=1031.582,202.326,-110.243,169.737,44.288,158.386
C05156=1031.589,202.574,-110.268,169.741,44.287,158.386
C05157=1031.595,202.824,-110.292,169.745,44.285,158.386
C05158=1031.601,203.072,-110.318,169.749,44.284,158.386
C05159=1031.607,203.320,-110.343,169.752,44.283,158.386
C05160=1031.612,203.570,-110.367,169.755,44.281,158.386
C05161=1031.619,203.818,-110.393,169.759,44.280,158.386
C05162=1031.625,204.067,-110.418,169.763,44.278,158.386
C05163=1031.651,205.115,-110.522,170.110,44.383,158.440
C05164=1031.661,205.472,-110.560,170.113,44.382,158.440
C05165=1031.670,205.830,-110.597,170.117,44.381,158.440
C05166=1031.679,206.187,-110.635,170.121,44.380,158.440
C05167=1031.690,206.543,-110.673,170.125,44.379,158.441
C05168=1031.697,206.792,-110.700,170.127,44.378,158.441
C05169=1031.703,207.040,-110.727,170.130,44.378,158.441
C05170=1031.710,207.289,-110.753,170.133,44.377,158.441
C05171=1031.716,207.537,-110.779,170.135,44.377,158.441
C05172=1031.723,207.786,-110.805,170.138,44.376,158.441
C05173=1031.730,208.035,-110.832,170.141,44.376,158.441
C05174=1031.736,208.283,-110.859,170.143,44.374,158.441
C05175=1031.743,208.532,-110.885,170.146,44.374,158.441
C05176=1031.750,208.780,-110.911,170.148,44.373,158.442
C05177=1031.757,209.028,-110.937,170.151,44.373,158.442
C05178=1031.763,209.278,-110.964,170.154,44.372,158.442
C05179=1031.770,209.526,-110.990,170.156,44.372,158.442
C05180=1031.777,209.774,-111.017,170.159,44.371,158.442
C05181=1031.783,210.023,-111.044,170.162,44.371,158.442
C05182=1031.790,210.271,-111.070,170.164,44.370,158.442
C05183=1031.797,210.520,-111.097,170.167,44.370,158.442
C05184=1031.803,210.768,-111.124,170.169,44.369,158.443
C05185=1031.810,211.017,-111.150,170.172,44.369,158.443
C05186=1031.817,211.265,-111.177,170.175,44.368,158.443
C05187=1031.823,211.514,-111.203,170.177,44.367,158.443
C05188=1031.830,211.762,-111.230,170.180,44.367,158.443
C05189=1031.837,212.011,-111.257,170.184,44.366,158.443
C05190=1031.843,212.259,-111.283,170.186,44.366,158.443
C05191=1031.850,212.508,-111.310,170.189,44.365,158.444
C05192=1031.857,212.756,-111.338,170.192,44.365,158.444
C05193=1031.863,213.005,-111.364,170.194,44.364,158.444
C05194=1031.870,213.253,-111.391,170.197,44.364,158.444
C05195=1031.877,213.502,-111.418,170.200,44.363,158.444
C05196=1031.883,213.750,-111.444,170.202,44.363,158.444
C05197=1031.890,213.999,-111.471,170.205,44.362,158.444
C05198=1031.897,214.248,-111.498,170.207,44.362,158.444
C05199=1031.903,214.495,-111.525,170.210,44.361,158.445
C05200=1031.910,214.744,-111.552,170.213,44.360,158.445
C05201=1031.916,214.993,-111.579,170.215,44.360,158.445
C05202=1031.923,215.241,-111.605,170.218,44.359,158.445
C05203=1031.930,215.489,-111.632,170.221,44.359,158.445
C05204=1031.937,215.738,-111.660,170.224,44.358,158.445
C05205=1031.944,215.987,-111.686,170.226,44.358,158.445
C05206=1031.950,216.235,-111.713,170.229,44.357,158.445
C05207=1031.957,216.483,-111.740,170.232,44.357,158.446
C05208=1031.964,216.732,-111.767,170.234,44.357,158.446
C05209=1031.971,216.980,-111.794,170.237,44.356,158.446
C05210=1031.977,217.229,-111.821,170.240,44.355,158.446
C05211=1031.984,217.477,-111.847,170.242,44.355,158.446
C05212=1031.991,217.726,-111.875,170.246,44.354,158.446
C05213=1031.998,217.975,-111.901,170.249,44.354,158.447
C05214=1032.004,218.222,-111.929,170.252,44.353,158.447
C05215=1032.011,218.471,-111.955,170.254,44.353,158.447
C05216=1032.017,218.719,-111.983,170.257,44.352,158.447
C05217=1032.025,218.968,-112.009,170.260,44.351,158.447
C05218=1032.031,219.217,-112.037,170.262,44.351,158.447
C05219=1032.037,219.465,-112.063,170.265,44.350,158.447
C05220=1032.047,219.828,-112.104,170.269,44.350,158.448
C05221=1032.057,220.190,-112.143,170.273,44.349,158.448
C05222=1032.067,220.553,-112.183,170.277,44.349,158.448
C05223=1032.076,220.915,-112.223,170.281,44.348,158.448
C05224=1032.082,221.164,-112.250,170.284,44.347,158.448
C05225=1032.090,221.413,-112.277,170.287,44.347,158.449
C05226=1032.096,221.661,-112.305,170.290,44.347,158.449
C05227=1032.103,221.910,-112.332,170.293,44.346,158.449
C05228=1032.109,222.158,-112.360,170.295,44.346,158.449
C05229=1032.116,222.406,-112.386,170.298,44.345,158.449
C05230=1032.123,222.655,-112.413,170.301,44.345,158.450
C05231=1032.129,222.903,-112.441,170.304,44.345,158.450
C05232=1032.136,223.152,-112.469,170.306,44.344,158.450
C05233=1032.143,223.400,-112.497,170.309,44.343,158.450
C05234=1032.150,223.649,-112.523,170.312,44.343,158.450
C05235=1032.156,223.897,-112.550,170.315,44.343,158.450
C05236=1032.163,224.145,-112.578,170.317,44.342,158.451
C05237=1032.169,224.394,-112.606,170.320,44.342,158.451
C05238=1032.176,224.643,-112.633,170.323,44.341,158.451
C05239=1032.183,224.891,-112.660,170.327,44.341,158.451
C05240=1032.190,225.139,-112.688,170.329,44.341,158.451
C05241=1032.196,225.388,-112.715,170.332,44.340,158.451
C05242=1032.203,225.636,-112.743,170.335,44.340,158.452
C05243=1032.209,225.885,-112.770,170.338,44.339,158.452
C05244=1032.216,226.133,-112.797,170.340,44.339,158.452
C05245=1032.223,226.381,-112.825,170.343,44.339,158.452
C05246=1032.230,226.630,-112.852,170.346,44.338,158.452
C05247=1032.236,226.878,-112.880,170.349,44.337,158.452
C05248=1032.243,227.126,-112.908,170.352,44.337,158.453
C05249=1032.250,227.375,-112.935,170.355,44.337,158.453
C05250=1032.257,227.624,-112.962,170.358,44.336,158.453
C05251=1032.264,227.872,-112.990,170.361,44.336,158.453
C05252=1032.270,228.121,-113.017,170.364,44.336,158.453
C05253=1032.277,228.369,-113.045,170.366,44.335,158.453
C05254=1032.284,228.617,-113.073,170.369,44.335,158.454
C05255=1032.290,228.865,-113.100,170.372,44.335,158.454
C05256=1032.296,229.114,-113.128,170.375,44.334,158.454
C05257=1032.303,229.362,-113.156,170.377,44.334,158.454
C05258=1032.310,229.610,-113.184,170.381,44.334,158.454
C05259=1032.317,229.858,-113.212,170.384,44.333,158.455
C05260=1032.323,230.107,-113.240,170.387,44.332,158.455
C05261=1032.330,230.355,-113.267,170.390,44.333,158.455
C05262=1032.337,230.604,-113.295,170.392,44.332,158.455
C05263=1032.343,230.852,-113.323,170.395,44.331,158.455
C05264=1032.350,231.100,-113.351,170.398,44.332,158.456
C05265=1032.357,231.349,-113.378,170.401,44.331,158.456
C05266=1032.363,231.598,-113.407,170.405,44.331,158.456
C05267=1032.369,231.846,-113.434,170.407,44.330,158.456
C05268=1032.376,232.094,-113.463,170.410,44.330,158.456
C05269=1032.383,232.342,-113.490,170.413,44.330,158.457
C05270=1032.390,232.591,-113.518,170.416,44.329,158.457
C05271=1032.396,232.839,-113.546,170.419,44.329,158.457
C05272=1032.402,233.088,-113.574,170.421,44.329,158.457
C05273=1032.409,233.336,-113.603,170.424,44.329,158.457
C05274=1032.416,233.584,-113.630,170.428,44.328,158.458
C05275=1032.423,233.833,-113.658,170.431,44.328,158.458
C05276=1032.432,234.188,-113.698,170.435,44.327,158.458
C05277=1032.442,234.542,-113.739,170.439,44.327,158.458
C05278=1032.452,234.898,-113.779,170.443,44.326,158.459
C05279=1032.461,235.254,-113.819,170.447,44.326,158.459
C05280=1032.468,235.501,-113.847,170.451,44.326,158.459
C05281=1032.474,235.750,-113.876,170.454,44.326,158.459
C05282=1032.480,235.999,-113.903,170.456,44.326,158.460
C05283=1032.487,236.246,-113.932,170.459,44.325,158.460
C05284=1032.494,236.495,-113.959,170.462,44.325,158.460
C05285=1032.501,236.743,-113.987,170.465,44.325,158.460
C05286=1032.507,236.991,-114.016,170.468,44.324,158.460
C05287=1032.514,237.240,-114.044,170.472,44.324,158.461
C05288=1032.521,237.488,-114.073,170.475,44.323,158.461
C05289=1032.528,237.737,-114.100,170.477,44.324,158.461
C05290=1032.534,237.986,-114.129,170.480,44.323,158.461
C05291=1032.541,238.233,-114.157,170.483,44.323,158.462
C05292=1032.548,238.482,-114.185,170.486,44.322,158.462
C05293=1032.555,238.730,-114.213,170.490,44.322,158.462
C05294=1032.560,238.978,-114.242,170.493,44.322,158.462
C05295=1032.567,239.226,-114.270,170.496,44.322,158.463
C05296=1032.575,239.475,-114.298,170.499,44.321,158.463
C05297=1032.582,239.723,-114.327,170.501,44.321,158.463
C05298=1032.588,239.972,-114.355,170.505,44.321,158.463
C05299=1032.595,240.220,-114.383,170.508,44.321,158.463
C05300=1032.601,240.468,-114.411,170.511,44.321,158.464
C05301=1032.608,240.716,-114.440,170.514,44.320,158.464
C05302=1032.615,240.964,-114.469,170.517,44.320,158.464
C05303=1032.621,241.214,-114.497,170.520,44.320,158.464
C05304=1032.628,241.461,-114.526,170.523,44.320,158.465
C05305=1032.634,241.710,-114.555,170.526,44.320,158.465
C05306=1032.641,241.958,-114.583,170.529,44.319,158.465
C05307=1032.647,242.206,-114.612,170.532,44.319,158.465
C05308=1032.654,242.454,-114.641,170.535,44.319,158.466
C05309=1032.660,242.703,-114.668,170.538,44.319,158.466
C05310=1032.667,242.952,-114.698,170.542,44.319,158.466
C05311=1032.674,243.199,-114.726,170.545,44.319,158.466
C05312=1032.680,243.448,-114.755,170.548,44.318,158.466
C05313=1032.687,243.696,-114.783,170.551,44.318,158.467
C05314=1032.693,243.944,-114.812,170.553,44.318,158.467
C05315=1032.701,244.193,-114.841,170.556,44.318,158.467
C05316=1032.707,244.441,-114.870,170.560,44.318,158.467
C05317=1032.714,244.689,-114.898,170.563,44.318,158.468
C05318=1032.720,244.937,-114.927,170.566,44.318,158.468
C05319=1032.726,245.185,-114.956,170.570,44.318,158.468
C05320=1032.733,245.434,-114.985,170.573,44.317,158.469
C05321=1032.739,245.682,-115.014,170.576,44.317,158.469
C05322=1032.746,245.930,-115.043,170.579,44.317,158.469
C05323=1032.753,246.178,-115.072,170.582,44.317,158.469
C05324=1032.759,246.426,-115.101,170.585,44.317,158.470
C05325=1032.766,246.675,-115.130,170.588,44.317,158.470
C05326=1032.772,246.923,-115.159,170.591,44.317,158.470
C05327=1032.779,247.171,-115.188,170.594,44.317,158.470
C05328=1032.785,247.419,-115.217,170.598,44.317,158.471
C05329=1032.792,247.668,-115.246,170.601,44.317,158.471
C05330=1032.798,247.916,-115.275,170.604,44.316,158.471
C05331=1032.805,248.165,-115.304,170.607,44.316,158.471
C05332=1032.814,248.513,-115.345,170.612,44.317,158.472
C05333=1032.823,248.863,-115.386,170.616,44.316,158.472
C05334=1032.832,249.212,-115.427,170.620,44.316,158.473
C05335=1032.842,249.562,-115.468,170.625,44.316,158.473
C05336=1032.849,249.810,-115.496,170.628,44.316,158.473
C05337=1032.855,250.058,-115.526,170.631,44.316,158.474
C05338=1032.862,250.307,-115.555,170.634,44.316,158.474
C05339=1032.868,250.555,-115.584,170.637,44.316,158.474
C05340=1032.875,250.803,-115.613,170.641,44.316,158.474
C05341=1032.881,251.052,-115.642,170.644,44.316,158.475
C05342=1032.889,251.299,-115.672,170.647,44.316,158.475
C05343=1032.895,251.547,-115.701,170.651,44.316,158.475
C05344=1032.902,251.796,-115.730,170.654,44.316,158.476
C05345=1032.908,252.044,-115.759,170.657,44.316,158.476
C05346=1032.914,252.292,-115.788,170.660,44.316,158.476
C05347=1032.922,252.540,-115.818,170.663,44.315,158.476
C05348=1032.928,252.788,-115.847,170.667,44.315,158.477
C05349=1032.935,253.036,-115.876,170.670,44.315,158.477
C05350=1032.942,253.285,-115.905,170.673,44.315,158.477
C05351=1032.948,253.533,-115.935,170.676,44.315,158.478
C05352=1032.955,253.781,-115.964,170.680,44.315,158.478
C05353=1032.962,254.029,-115.993,170.683,44.315,158.478
C05354=1032.968,254.277,-116.022,170.686,44.315,158.478
C05355=1032.975,254.526,-116.052,170.690,44.315,158.479
C05356=1032.982,254.774,-116.081,170.693,44.315,158.479
C05357=1032.988,255.023,-116.110,170.696,44.315,158.479
C05358=1032.995,255.270,-116.140,170.699,44.314,158.480
C05359=1033.003,255.519,-116.169,170.702,44.314,158.480
C05360=1033.009,255.767,-116.198,170.706,44.314,158.480
C05361=1033.016,256.015,-116.228,170.709,44.314,158.480
C05362=1033.022,256.263,-116.257,170.712,44.315,158.481
C05363=1033.029,256.512,-116.287,170.716,44.315,158.481
C05364=1033.036,256.759,-116.316,170.719,44.315,158.481
C05365=1033.042,257.008,-116.346,170.722,44.315,158.482
C05366=1033.050,257.255,-116.375,170.725,44.315,158.482
C05367=1033.057,257.504,-116.404,170.729,44.315,158.482
C05368=1033.063,257.752,-116.434,170.733,44.314,158.483
C05369=1033.070,258.001,-116.463,170.736,44.314,158.483
C05370=1033.077,258.248,-116.493,170.739,44.314,158.483
C05371=1033.083,258.497,-116.523,170.743,44.314,158.483
C05372=1033.090,258.745,-116.552,170.746,44.314,158.484
C05373=1033.098,258.993,-116.581,170.749,44.314,158.484
C05374=1033.104,259.240,-116.611,170.753,44.314,158.484
C05375=1033.111,259.489,-116.640,170.756,44.314,158.485
C05376=1033.118,259.738,-116.670,170.759,44.314,158.485
C05377=1033.124,259.986,-116.699,170.762,44.314,158.485
C05378=1033.132,260.234,-116.730,170.766,44.314,158.486
C05379=1033.138,260.482,-116.759,170.769,44.314,158.486
C05380=1033.146,260.730,-116.788,170.773,44.314,158.486
C05381=1033.152,260.978,-116.817,170.776,44.314,158.487
C05382=1033.159,261.226,-116.847,170.780,44.314,158.487
C05383=1033.166,261.474,-116.877,170.783,44.314,158.487
C05384=1033.173,261.723,-116.906,170.786,44.314,158.487
C05385=1033.179,261.971,-116.937,170.790,44.314,158.488
C05386=1033.185,262.219,-116.967,170.793,44.314,158.488
C05387=1033.193,262.467,-116.997,170.796,44.314,158.488
C05388=1033.201,262.815,-117.038,170.802,44.315,158.489
C05389=1033.211,263.163,-117.081,170.806,44.315,158.489
C05390=1033.221,263.511,-117.123,170.811,44.315,158.490
